TYPE ST_CoordinateGantryAxisEnable :
STRUCT
    {attribute 'pytmc' := '
        pv: bEnable
        io: i
        field: DESC Set false to prevent this function block from allowing the motors to enable.
    '}
    bEnable: BOOL; // Set false to prevent this function block from allowing the motors to enable.
    {attribute 'pytmc' := '
        pv: bLeaderDriveReady
        io: i
        field: DESC Intended to be linked to the leader drive ready status.
    '}
    bLeaderDriveReady AT %I*: BOOL; // Intended to be linked to the leader drive ready status.
    {attribute 'pytmc' := '
        pv: bFollowDriveReady
        io: i
        field: DESC Intended to be linked to the follow drive ready status.
    '}
    bFollowDriveReady AT %I*: BOOL; // Intended to be linked to the follow drive ready status.
    tTimeout: TIME := T#5s; // Timeout before giving up on a state.
    {attribute 'pytmc' := '
        pv: eState
        io: i
        field: DESC Present enable sequence state.
    '}
    eState: E_GantryEnableState; // Present enable sequence state.
END_STRUCT
END_TYPE

// ---- DUTs/ST_GarageSlot.TcDUT

TYPE ST_GarageSlot EXTENDS ST_SampleSlot :
(*
    Represents a slot in the SDS garage.
*)
STRUCT
    {attribute 'pytmc' := '
        pv: fYPos
        io: io
        field: DESC The y-position of the garage, in units of mm, which corresponds to the slot being approximately level with the transfer arm.
    '}
    fYPos: REAL;
    {attribute 'pytmc' := '
        pv: fDeg
        io: io
        field: DESC The angular position of the slot in the garage in units of degrees.
    '}
    fDeg: REAL;
END_STRUCT
END_TYPE

// ---- DUTs/ST_BoundedValue.TcDUT

TYPE ST_BoundedValue :
STRUCT
    {attribute 'pytmc' := '
        pv: fIn
        io: io
        field: DESC The input value before bounds are applied.
    '}
    fIn    : LREAL; // The input value before bounds are applied.
    {attribute 'pytmc' := '
        pv: fMax
        io: io
        field: DESC The maximum bound for the output value.
    '}
    fMax   : LREAL; // The maximum bound for the output value.
    {attribute 'pytmc' := '
        pv: fMin
        io: io
        field: DESC The minimum bound for the output value.
    '}
    fMin   : LREAL; // The minimum bound for the output value.
    {attribute 'pytmc' := '
        pv: fOut
        io: i
        field: DESC The output value after bounds are applied.
    '}
    fOut   : LREAL; // The output value after bounds are applied.
    {attribute 'pytmc' := '
        pv: bMaxLim
        io: i
        field: DESC TRUE if the output value has been limited by the upper bound.
    '}
    bMaxLim: BOOL; // TRUE if the output value has been limited by the upper bound.
    {attribute 'pytmc' := '
        pv: bMinLim
        io: i
        field: DESC TRUE if the output value has been limited by the lower bound.
    '}
    bMinLim: BOOL; // TRUE if the output value has been limited by the lower bound.
END_STRUCT
END_TYPE

// ---- DUTs/ST_DiffractometerSlot.TcDUT

TYPE ST_DiffractometerSlot EXTENDS ST_SampleSlot :
(*
    Represents a slot in the SDS garage.
*)
STRUCT
    {attribute 'pytmc' := '
        pv: fYPos
        io: io
        field: DESC The y-position of the garage, in units of mm, which corresponds to the slot being approximately level with the transfer arm.
    '}
    fYPos: REAL;
    {attribute 'pytmc' := '
        pv: fDeg
        io: io
        field: DESC The angular position of the slot in the garage in units of degrees.
    '}
    fDeg: REAL;
END_STRUCT
END_TYPE

// ---- DUTs/ST_MultiLeaderMotionCoupling.TcDUT

TYPE ST_MultiLeaderMotionCoupling :
STRUCT
    {attribute 'pytmc' := '
        pv: bEnable
        io: io
        field: DESC Set and hold TRUE to allow the axis to run in multi-leader mode.
    '}
    bEnable: BOOL;

    {attribute 'pytmc' := '
        pv: bReset
        io: io
        field: DESC Set and release TRUE to fully reset errors and state machine.
    '}
    bReset: BOOL;

    {attribute 'pytmc' := '
        pv: bBusy
        io: i
        field: DESC TRUE indicates state machine running and not in error state.
    '}
    bBusy: BOOL;

    {attribute 'pytmc' := '
        pv: sStatusMsg
        io: i
        field: DESC String used to give helpful messages.
    '}
    sStatusMsg: T_MaxString;

    // Ex: TIID^Device 2 (EtherCAT)^B950-233-WALL-S-R01-DRL-01^EL7047_02_11^STM Status^Status^Ready
    {attribute 'pytmc' := '
        pv: bFollowerDriveReady
        io: i
        field: DESC Linked to the ready status of the drive.
    '}
    bFollowerDriveReady AT %I*: BOOL; // Link to the ready status of the drive

    {attribute 'pytmc' := '
        pv: bUseDynamicLimits
        io: io
        field: DESC Set AND hold TRUE to enable dynamic limits to acc, vel, AND pos.
    '}
    bUseDynamicLimits: BOOL;

    {attribute 'pytmc' := '
        pv: fTargetAcc
        io: io
        field: DESC The target acceleration.
    '}
    fTargetAcc: LREAL; // Set in software to allow axis to target an acceleration based on multiple leaders.

    {attribute 'pytmc' := '
        pv: fTargetVel
        io: io
        field: DESC The target velocity.
    '}
    fTargetVel: LREAL; // Set in software to allow axis to target a velocity based on multiple leaders.

    {attribute 'pytmc' := '
        pv: fTargetPos
        io: io
        field: DESC The target position.
    '}
    fTargetPos: LREAL; // Set in software to allow axis to target a position based on multiple leaders.

    {attribute 'pytmc' := '
        pv: fPosDelta
        io: i
        field: DESC Target position minus position.
    '}
    fPosDelta : LREAL; // Difference between current position and target position.

    {attribute 'pytmc' := '
        pv: fTTGain
        io: io
        field: DESC Target tracking gain.
    '}
    fTargetTrackingGain: LREAL := 1; // Gain used to tune target tracking when within target position window.

    {attribute 'pytmc' := '
        pv: fHaltPos
        io: i
        field: DESC Position at which axis halted.
    '}
    fHaltPos: LREAL; // Position at which halt is called. Allows for centering deadband.

    {attribute 'pytmc' := 'pv: stAcc'}
    stAcc: ST_BoundedValue;

    {attribute 'pytmc' := 'pv: stVel'}
    stVel: ST_BoundedValue;

    {attribute 'pytmc' := 'pv: stPos'}
    stPos: ST_BoundedValue;

    {attribute 'pytmc' := '
        pv: nDir
        io: i
        field: DESC Internally calculated direction value for external setpoint generator.
    '}
    nDir: DINT;

    {attribute 'pytmc' := '
        pv: bError
        io: i
        field: DESC TRUE if an error is active.
    '}
    bError: BOOL;

    {attribute 'pytmc' := '
        pv: sErrorMsg
        io: i
        field: DESC Displays error message relevant to the active error. Empty otherwise.
    '}
    sErrorMsg: T_MaxString;

    {attribute 'pytmc' := '
        pv: sErrorHelp
        io: i
        field: DESC Displays additional help for the active rror. Empty otherwise.
    '}
    sErrorHelp: T_MaxString;

    {attribute 'pytmc' := '
        pv: eState
        io: i
        field: DESC Records the current state of the multi-leader function block.
    '}
    eState: E_MultiLeaderMotionCoupling;
END_STRUCT
END_TYPE

// ---- DUTs/ST_SampleSlot.TcDUT

TYPE ST_SampleSlot :
(*
    Represents a general slot for a sample puck.
*)
STRUCT
    {attribute 'pytmc' := '
        pv: eState
        io: io
        field: DESC Enumeration of possible states for a slot in the sample delivery system. (empty, full, or disabled)
    '}
    eState: E_SampleSlotStates;
    {attribute 'pytmc' := '
        pv: sTag
        io: i
        field: DESC A two character identifier for the slot. e.g., T1, B3, etc...
    '}
    sTag: STRING;
    {attribute 'pytmc' := '
        pv: sDesc
        io: io
        field: DESC If the slot is in the full state, this value is supposed to describe what is in the slot.
    '}
    sDesc: T_MaxString;
END_STRUCT
END_TYPE

// ---- DUTs/ST_SDS.TcDUT

TYPE ST_SDS :
(*
    Structure to represent the data used for the sample delivery system that is not
    needed to be persistent.
*)
STRUCT
    {attribute 'pytmc' := '
        pv: Initialized
        io: i
        field: DESC TRUE if the non-persistent data has been initialized. FALSE if it has not.
    '}
    bInitialized: BOOL;

    {attribute 'pytmc' := '
        pv: Enable
        io: io
        field: DESC TRUE to enable SDS system. FALSE to disable.
    '}
    bEnable : BOOL := TRUE;

    {attribute 'pytmc' := '
        pv: Maint
        io: io
        field: DESC TRUE if in maintenance mode. FALSE if NOT.
    '}
    bMaint: BOOL;

    {attribute 'pytmc' := '
        pv: Error
        io: i
        field: DESC TRUE if an error is active. FALSE if not.
    '}
    bError : BOOL;

    {attribute 'pytmc' := '
        pv: ErrorMsg
        io: i
        field: DESC Error message to help describe the active error.
    '}
    sErrorMsg : T_MaxString;

    {attribute 'pytmc' := '
        pv: Success
        io: i
        field: DESC TRUE if successfully completed state machine step.
    '}
    bSuccess : BOOL;

    // Variables used for homing
    {attribute 'pytmc' := '
        pv: HomeReq
        io: i
        field: DESC TRUE if homing is required for the sample transfer arm.
    '}
    bHomingRequired : BOOL := TRUE;
    tHomingRequiredTimeoutTime : TIME := T#1h;
    tonHomingRequiredTimeout : TON;
    tonHomingStateTimeout : TON;
    nHomingState : INT := 0;
    {attribute 'pytmc' := '
        pv: MinHomeReq
        io: i
        field: DESC Minutes until homing is required again for the sample transfer arm.
    '}
    fMinUntilHomingRequired: REAL;

    {attribute 'pytmc' := '
        pv: FaceState
        io: i
        field: DESC Enum to describe which way the sample garage should face.
    '}
    eFaceState: E_SDSFaceState;

    {attribute 'pytmc' := '
        pv: FacePortOffset
        io: io
        field: DESC Degree offset when trying to face the side port.
    '}
    fFacePortOffset: REAL := 90; // degree offset when trying to face the side port.

    // Transfer Arm State Positioner
    stTransferArmHEpicsToPlc: ST_StateEpicsToPlc;
    stTransferArmHPlcToEpics: ST_StatePlcToEpics;

    {attribute 'pytmc' := '
      pv: ArmHStateGet
      io: i
    '}
    eTransferArmHStateGet: E_SDSTransferArmHStates; // get state enum for transfer arm horizontal position states.

    {attribute 'pytmc' := '
      pv: ArmHStateSet
      io: io
    '}
    eTransferArmHStateSet: E_SDSTransferArmHStates; // set state enum for transfer arm horizontal position states.

    astTransferArmHPosState: ARRAY[1..GeneralConstants.MAX_STATES] OF ST_PositionState;
    {attribute 'pytmc' := '
        pv: ARMH:PS1D
        field: DESC Position State 1D used for transfer arm horizontal position states.
    '}
    fbTransferArmHPos1D: FB_PositionState1D; // Position State 1D used for transfer arm horizontal position states.

    // Transfer Arm State Positioner
    stTransferArmREpicsToPlc: ST_StateEpicsToPlc;
    stTransferArmRPlcToEpics: ST_StatePlcToEpics;

    {attribute 'pytmc' := '
      pv: ArmRStateGet
      io: i
    '}
    eTransferArmRStateGet: E_SDSTransferArmRStates; // get state enum for transfer arm rotational position states.

    {attribute 'pytmc' := '
      pv: ArmRStateSet
      io: io
    '}
    eTransferArmRStateSet: E_SDSTransferArmRStates; // set state enum for transfer arm rotational position states.

    astTransferArmRPosState: ARRAY[1..GeneralConstants.MAX_STATES] OF ST_PositionState;
    {attribute 'pytmc' := '
        pv: ARMR:PS1D
        field: DESC Position State 1D used for transfer arm rotational position states.
    '}
    fbTransferArmRPos1D: FB_PositionState1D; // Position State 1D used for transfer arm rotational position states.

    // Garage Y State Positioner
    stGarageYEpicsToPlc: ST_StateEpicsToPlc;
    stGarageYPlcToEpics: ST_StatePlcToEpics;

    {attribute 'pytmc' := '
      pv: GarYStateGet
      io: i
    '}
    eGarageYStateGet: E_SDSGarageYStates; // get state enum for garage y and rotational position states.

    {attribute 'pytmc' := '
      pv: GarYStateSet
      io: io
    '}
    eGarageYStateSet: E_SDSGarageYStates; // set state enum for garage y and rotational position states.

    astGarageYPosState: ARRAY[1..GeneralConstants.MAX_STATES] OF ST_PositionState;

    {attribute 'pytmc' := '
        pv: GARY:PS1D
        field: DESC Position State 1D used for garage y-position.
    '}
    fbGarageYPos1D: FB_PositionState1D; // Position State 1D used for garage y-position.

    // Garage R State Positioner
    stGarageREpicsToPlc: ST_StateEpicsToPlc;
    stGarageRPlcToEpics: ST_StatePlcToEpics;

    {attribute 'pytmc' := '
      pv: GarRStateGet
      io: i
    '}
    eGarageRStateGet: E_SDSGarageRStates; // get state enum for garage y and rotational position states.

    {attribute 'pytmc' := '
      pv: GarRStateSet
      io: io
    '}
    eGarageRStateSet: E_SDSGarageRStates; // set state enum for garage y and rotational position states.

    astGarageRPosState: ARRAY[1..GeneralConstants.MAX_STATES] OF ST_PositionState;

    {attribute 'pytmc' := '
        pv: GARR:PS1D
        field: DESC Position State 1D used for garage rotation..
    '}
    fbGarageRPos1D: FB_PositionState1D; // Position State 1D used for garage rotation.

    {attribute 'pytmc' := '
        pv: State
        field: DESC Present state for sample delivery system.
    '}
    eState : E_SDSState;

    {attribute 'pytmc' := '
        pv: SubState
        field: DESC Present sub-state for sample delivery system.
    '}
    eSubState : E_SDSSubState;

    {attribute 'pytmc' := '
        pv: SeqState
        field: DESC Present sequence state for sample delivery system.
    '}
    eSeqState: E_SDSSeqState;

    {attribute 'pytmc' := '
        pv: SecRemaining
        field: DESC Seconds remaining before current sequence step times out.
    '}
    fSecRemaining: REAL;

    {attribute 'pytmc' := '
        pv: StatusMsg
        field: DESC Status message.
    '}
    sStatusMsg: T_MaxString;

    // Booleans to track what is currently possible to do.

    {attribute 'pytmc' := '
        pv: GarLoadable
        io: i
        field: DESC True if it is currently possible to load a garage slot. False if all garage slots are full or disabled.
    '}
    bGarageLoadable : BOOL;

    {attribute 'pytmc' := '
        pv: GarUnloadable
        io: i
        field: DESC True if it is currently possible to unload a garage slot. False if all garage slots are empty or disabled.
    '}
    bGarageUnloadable : BOOL;

    {attribute 'pytmc' := '
        pv: ArmLoadable
        io: i
        field: DESC True if it is currently possible to load the transfer arm slot. False if the transfer arm slot is full or disabled.
    '}
    bTransferArmLoadable : BOOL;

    {attribute 'pytmc' := '
        pv: ArmUnloadable
        io: i
        field: DESC True if it is currently possible to unload the transfer arm slot. False if the transfer arm slot is empty or disabled.
    '}
    bTransferArmUnloadable : BOOL;

    {attribute 'pytmc' := '
        pv: DiffLoadable
        io: i
        field: DESC True if it is currently possible to load the diffractometer slot. False if the diffractometer slot is full or disabled.
    '}
    bDiffractometerLoadable : BOOL;

    {attribute 'pytmc' := '
        pv: DiffUnloadable
        io: i
        field: DESC True if it is currently possible to unload the diffractometer slot. False if the diffractoemter slot is empty or disabled.
    '}
    bDiffractometerUnloadable : BOOL;

    {attribute 'pytmc' := 'pv: Sel'}
    stUISelect : ST_UISelect;

    tonForwardHomingLimit: TON;

    stGarageYStage : REFERENCE TO ST_MotionStage;
    stGarageRStage : REFERENCE TO ST_MotionStage;
    stTransferArmHStage : REFERENCE TO ST_MotionStage;
    stTransferArmRStage : REFERENCE TO ST_MotionStage;

    eDiffXStateGet : REFERENCE TO E_DiffState;
    eDiffXStateSet : REFERENCE TO E_DiffState;
    stDiffXStage : REFERENCE TO ST_MotionStage;

    eDiffYStateGet : REFERENCE TO E_DiffState;
    eDiffYStateSet : REFERENCE TO E_DiffState;
    stDiffYStage : REFERENCE TO ST_MotionStage;

    eDiffZStateGet : REFERENCE TO E_DiffState;
    eDiffZStateSet : REFERENCE TO E_DiffState;
    stDiffZStage : REFERENCE TO ST_MotionStage;

    eDiff2ThetaYStateGet : REFERENCE TO E_DiffState;
    eDiff2ThetaYStateSet : REFERENCE TO E_DiffState;
    stDiff2ThetaYStage : REFERENCE TO ST_MotionStage;

    eDiffPhiStateGet : REFERENCE TO E_DiffState;
    eDiffPhiStateSet : REFERENCE TO E_DiffState;
    stDiffPhiStage : REFERENCE TO ST_MotionStage;

    eDiffChiStateGet : REFERENCE TO E_DiffState;
    eDiffChiStateSet : REFERENCE TO E_DiffState;
    stDiffChiStage : REFERENCE TO ST_MotionStage;

    eDiff2ThetaStateGet : REFERENCE TO E_DiffState;
    eDiff2ThetaStateSet : REFERENCE TO E_DiffState;
    stDiff2ThetaStage : REFERENCE TO ST_MotionStage;

    eDiffThetaStateGet : REFERENCE TO E_DiffState;
    eDiffThetaStateSet : REFERENCE TO E_DiffState;
    stDiffThetaStage : REFERENCE TO ST_MotionStage;

    {attribute 'pytmc' := '
        pv: GarAboveColl
        io: i
        field: DESC True if garage above collision height.
    '}
    bGarageAboveCollisionHeight : BOOL;

    {attribute 'pytmc' := '
        pv: TAHHomeState
        io: i
        field: DESC Transfer arm horizontal homing state.
    '}
    eTransferArmHHomingState : E_SDSHomingState;

    {attribute 'pytmc' := '
        pv: TARHomeState
        io: i
        field: DESC Transfer arm rotational homing state.
    '}
    eTransferArmRHomingState : E_SDSHomingState;

    {attribute 'pytmc' := '
        pv: GarRHomeState
        io: i
        field: DESC Garage rotational homing state.
    '}
    eGarageRHomingState : E_SDSHomingState;

    {attribute 'pytmc' := '
        pv: GarRotSpeed
        io: i
        field: DESC Garage rotational speed.
    '}
    fGarageRotationSpeed : LREAL := 10.0;

    {attribute 'pytmc' := '
        pv: TARotSpeed
        io: i
        field: DESC Garage rotational speed.
    '}
    fTransferArmRotationSpeed : LREAL := 10.0;

    {attribute 'pytmc' := '
        pv: GarRotClearancePos
        io: i
        field: DESC Garage rotational position to avoid collision with loaded transfer arm when moving up and down.
    '}
    fGarageRotationClearancePos : LREAL;

    {attribute 'pytmc' := '
        pv: LoadingSel
        io: i
        field: DESC True if loading from port.
    '}
    bLoadingSelected : BOOL;

    {attribute 'pytmc' := '
        pv: UnloadingSel
        io: i
        field: DESC True if unloading from port.
    '}
    bUnloadingSelected : BOOL;

    {attribute 'pytmc' := '
        pv: NumGarSlots
        io: i
        field: DESC Number of garage sample slots.
    '}
    nGarageSlots : UINT := 12;

    {attribute 'pytmc' := '
        pv: SelGarSlot
        io: i
        field: DESC Selected garage slot for loading/unloading.
    '}
    eSelectedGarageSlot : E_SDSGarageYStates;
END_STRUCT
END_TYPE

// ---- DUTs/ST_SDSPersistent.TcDUT

TYPE ST_SDSPersistent :
(*
    Structure to represent the data used for the sample delivery system that is
    needed to be persistent.
*)
STRUCT
    {attribute 'pytmc' := '
        pv: bInitialized
        io: i
        field: DESC TRUE if the persistent data has been initialized. FALSE if it has not.
    '}
    bInitialized: BOOL;

    {attribute 'pytmc' := 'pv: Garage:Slot'}
    astGarageSlot: ARRAY[E_SDSGarageYStates.T1..E_SDSGarageYStates.B4] OF ST_GarageSlot;

    {attribute 'pytmc' := 'pv: Transfer:Slot'}
    stTransferArmSlot: ST_TransferSlot;

    {attribute 'pytmc' := 'pv: Diff:Slot'}
    stDiffractometerSlot: ST_DiffractometerSlot;

    {attribute 'pytmc' := '
        pv: GarHSafeFromCol
        io: i
        field: DESC Height at which garage consider safe from collisions.
    '}
    fGarageHeightSafeFromCollision : LREAL := -10;

    {attribute 'pytmc' := '
        pv: GarRClearOff
        io: i
        field: DESC Garage rotational offset for clearance when moving up and down with loading transfer arm.
    '}
    fGarageRotationClearanceOffset : LREAL := 45;
END_STRUCT
END_TYPE

// ---- DUTs/ST_TransferSlot.TcDUT

TYPE ST_TransferSlot EXTENDS ST_SampleSlot :
(*
    Represents a slot in the SDS transfer arm.
*)
STRUCT
END_STRUCT
END_TYPE

// ---- DUTs/ST_UISelect.TcDUT

TYPE ST_UISelect :
STRUCT
    // Booleans to allow operator to choose what they want to do.
    {attribute 'pytmc' := '
        pv: Load
        io: io
        field: DESC Write True to command a loading sequence.
    '}
    bLoad: BOOL;

    {attribute 'pytmc' := '
        pv: Unload
        io: io
        field: DESC Write True to command a unloading sequence.
    '}
    bUnload: BOOL;

    {attribute 'pytmc' := '
        pv: ManualControl
        io: io
        field: DESC Write True to command manual control.
    '}
    bManualControl : BOOL;

    {attribute 'pytmc' := '
        pv: ExitManualControl
        io: io
        field: DESC Write True to command exit manual control.
    '}
    bExitManualControl : BOOL;

    {attribute 'pytmc' := '
        pv: LoadArmFromGar
        io: io
        field: DESC Write True to command load arm from garage.
    '}
    bLoadArmFromGarage : BOOL;

    {attribute 'pytmc' := '
        pv: UnloadArmToGar
        io: io
        field: DESC Write True to command unload arm from garage.
    '}
    bUnloadArmToGarage : BOOL;

    {attribute 'pytmc' := '
        pv: LoadGarFromPort
        io: io
        field: DESC Write True to command load garage from port.
    '}
    bLoadGarageFromPort : BOOL;

    {attribute 'pytmc' := '
        pv: UnloadGarFromPort
        io: io
        field: DESC Write True to command load garage from port.
    '}
    bLoadUnloadGarageFromPort : BOOL;

    {attribute 'pytmc' := '
        pv: LoadDiffFromArm
        io: io
        field: DESC Write True to command load diffractometer from arm.
    '}
    bLoadDiffractometerFromArm : BOOL;

    {attribute 'pytmc' := '
        pv: UnloadDiffToArm
        io: io
        field: DESC Write True to command unload diffractometer to arm.
    '}
    bUnloadDiffractometerToArm : BOOL;

    {attribute 'pytmc' := '
        pv: HomeArm
        io: io
        field: DESC Write True to command home transfer arm.
    '}
    bHomeTransferArm : BOOL;

    {attribute 'pytmc' := '
        pv: HomeGar
        io: io
        field: DESC Write True to command home garage.
    '}
    bHomeGarage : BOOL;

    {attribute 'pytmc' := '
        pv: GarSlot
        io: io
        field: DESC Select garage slot to unload or load.
    '}
    eGarageSlot : E_SDSGarageYStates;

    {attribute 'pytmc' := '
        pv: Proceed
        io: io
        field: DESC Write True to proceed to next sequence step, if applicable.
    '}
    bProceed: BOOL;

    {attribute 'pytmc' := '
        pv: Retry
        io: io
        field: DESC Write True when prompted to retry a defined previous step, if applicable.
    '}
    bRetry: BOOL;

    {attribute 'pytmc' := '
        pv: Cancel
        io: io
        field: DESC TRUE to cancel next sequence step.
    '}
    bCancel: BOOL;

    {attribute 'pytmc' := '
        pv: TextInput
        io: io
        field: DESC General purpose text input field.
    '}
    sTextInput: T_MaxString;
END_STRUCT
END_TYPE

// ---- Version/Global_Version.TcGVL
{attribute 'TcGenerated'}
{attribute 'no-analysis'}
{attribute 'linkalways'}
// This function has been automatically generated from the project information.
VAR_GLOBAL CONSTANT
    {attribute 'const_non_replaced'}
    stLibVersion_qrix_motion : ST_LibVersion := (iMajor := 0, iMinor := 4, iBuild := 0, iRevision := 0, nFlags := 1, sVersion := '0.4.0');
END_VAR

// ---- GVLs/GVL_EPS.TcGVL

VAR_GLOBAL
    {attribute 'pytmc' := 'pv: QRIX:SA:ESTOP_RST'}
    bResetIClk: BOOL;
    {attribute 'pytmc' := 'pv: QRIX:SA:ESTOP'}
    {attribute 'TcLinkTo' := 'TIIB[Rack#1A-02 SFIN (EL1918)]^StandardInputs^Standard Out Var 18'}
    bESTOP AT %I*: BOOL;

    {attribute 'TcLinkTo' := 'TIIB[Rack#2B-05 SV_AIR (EL2004)]^Channel 1^Output'}
    {attribute 'pytmc' := 'pv: QRIX:SA:SV1'}
    bOpenSV1 AT %Q*: BOOL;
    {attribute 'TcLinkTo' := 'TIIB[Rack#2B-05 SV_AIR (EL2004)]^Channel 2^Output'}
    {attribute 'pytmc' := 'pv: QRIX:SA:SV2'}
    bOpenSV2 AT %Q*: BOOL;

    {attribute 'TcLinkTo' := 'TIIB[Rack#1C_ServoDR (NCR-HD Series)]^260th receive PDO Mapping^Positive torque limit value'}
    iServoTorqueLimitPositive AT %Q*: UINT;

    {attribute 'TcLinkTo' := 'TIIB[Rack#1C_ServoDR (NCR-HD Series)]^260th receive PDO Mapping^Negative torque limit value'}
    iServoTorqueLimitNegative AT %Q*: UINT;

END_VAR

// ---- GVLs/GVL_Interface.TcGVL

{attribute 'qualified_only'}
VAR_GLOBAL

    (*I/O Outputs to QRIX Vacuum PLC*)

    {attribute 'TcLinkTo' :=  'TIID^Device 2 (EtherCAT)^B950-233-R03-DRL-01 (EK1200)^Term 141 (EL6692)^IO Outputs^QRIX_MOT_SDS_MMS_H_RAW_ENC_CNTS
    '}
    QRIX_MOT_SDS_MMS_H_RAW_ENC_CNTS AT %Q* : UINT;

    {attribute 'TcLinkTo' :=  'TIID^Device 2 (EtherCAT)^B950-233-R03-DRL-01 (EK1200)^Term 141 (EL6692)^IO Outputs^QRIX_MOT_SDS_MMS_H_FORWARD_EN
    '}
    QRIX_MOT_SDS_MMS_H_FORWARD_EN AT %Q* : BOOL;

    {attribute 'TcLinkTo' :=  'TIID^Device 2 (EtherCAT)^B950-233-R03-DRL-01 (EK1200)^Term 141 (EL6692)^IO Outputs^QRIX_MOT_SDS_MMS_H_BACKWARD_EN
    '}
    QRIX_MOT_SDS_MMS_H_BACKWARD_EN AT %Q* : BOOL;

    (*I/O Inputs from QRIX Vacuum PLC*)

    {attribute 'TcLinkTo' :=  'TIID^Device 2 (EtherCAT)^B950-233-R03-DRL-01 (EK1200)^Term 141 (EL6692)^IO Inputs^QRIX_VAC_VGC_03_OPEN_LIMIT_SWITCH
    '}
    QRIX_VAC_VGC_03_OPEN_LIMIT_SWITCH AT %I* : BOOL;

    {attribute 'TcLinkTo' :=  'TIID^Device 2 (EtherCAT)^B950-233-R03-DRL-01 (EK1200)^Term 141 (EL6692)^IO Inputs^QRIX_VAC_VGC_03_CLOSED_LIMIT_SWITCH
    '}
    QRIX_VAC_VGC_03_CLOSED_LIMIT_SWITCH AT %I* : BOOL;
    {attribute 'TcLinkTo' :=  'TIID^Device 2 (EtherCAT)^B950-233-R03-DRL-01 (EK1200)^Term 141 (EL6692)^IO Inputs^QRIX_VAC_VGC_03_OP_CMD
    '}
    QRIX_VAC_VGC_03_OP_CMD AT %I* : BOOL;

    {attribute 'TcLinkTo' :=  'TIID^Device 2 (EtherCAT)^B950-233-R03-DRL-01 (EK1200)^Term 141 (EL6692)^IO Inputs^QRIX_VAC_VGC_03_CL_CMD
    '}
    QRIX_VAC_VGC_03_CL_CMD AT %I* : BOOL;
END_VAR

// ---- GVLs/GVL_PMPS.TcGVL

{attribute 'qualified_only'}
VAR_GLOBAL
    {attribute 'pytmc' := 'pv: PLC:QRIX:MOTION:ARB'}
    fbArbiter: FB_Arbiter(1);
    {attribute 'pytmc' := 'pv: PLC:QRIX:MOTION:FFO:01'}
    {attribute 'TcLinkTo' := '.q_xFastFaultOut:=TIIB[PMPS_FFO]^Channel 1^Output'}
    fbFastFaultOutput1: FB_HardwareFFOutput := (bAutoReset := TRUE, i_sNetID:='172.21.92.73.1.1');
    {attribute 'pytmc' := 'pv: PLC:QRIX:MOTION:FFO:02'}
    {attribute 'TcLinkTo' := '.q_xFastFaultOut:=TIIB[PMPS_FFO]^Channel 2^Output'}
    fbFastFaultOutput2: FB_HardwareFFOutput := (bAutoReset := TRUE, i_sNetID:='172.21.92.73.1.1');
END_VAR

// ---- GVLs/GVL_Sensor.TcGVL

{attribute 'qualified_only'}
VAR_GLOBAL
    {attribute 'pytmc' := '
        pv: QRIX:SA:FLOATING
        io: i
    '}
    bFloating: BOOL;

    // YDF1
    {attribute 'pytmc' := '
        pv: QRIX:SA:DDS:YDF1
        io: i
    '}
    {attribute 'TcLinkTo' := '	.iRawCnts	:= TIIB[Rack#2D LinearGaugeAmp (SC-HG1-ETC)]^Process Data(In)  TxPDO-Map^Response Data Unit1'}
    stYDF1: DUT_SensorHGS;
    nYDF1 AT %Q*: UDINT;

    // YDF2
    {attribute 'pytmc' := '
        pv: QRIX:SA:DDS:YDF2
        io: i
    '}
    {attribute 'TcLinkTo' := '	.iRawCnts	:= TIIB[Rack#2D LinearGaugeAmp (SC-HG1-ETC)]^Process Data(In)  TxPDO-Map^Response Data Unit2'}
    stYDF2: DUT_SensorHGS;
    nYDF2 AT %Q*: UDINT;

    // YDF3
    {attribute 'pytmc' := '
        pv: QRIX:SA:DDS:YDF3
        io: i
    '}
    {attribute 'TcLinkTo' := '	.iRawCnts	:= TIIB[Rack#2D LinearGaugeAmp (SC-HG1-ETC)]^Process Data(In)  TxPDO-Map^Response Data Unit3'}
    stYDF3: DUT_SensorHGS;
    nYDF3 AT %Q*: UDINT;

    // Height difference btw granite shelf and detector frame.
    {attribute 'pytmc' := '
        pv: QRIX:SA:DDS:HDF
        io: i
    '}
    {attribute 'TcLinkTo' := '	.iRawCnts	:= TIIB[Rack#2D LinearGaugeAmp (SC-HG1-ETC)]^Process Data(In)  TxPDO-Map^Response Data Unit4'}
    stHDF: DUT_SensorHGS;

    // Granite TiltZ : Pitch
    {attribute 'pytmc' := '
        pv: QRIX:GS:INM:Z
        io: i
    '}
    {attribute 'TcLinkTo' := '	.iRawCnts	:= TIIB[Rack#2B-03 AI_TiltSensor (EL3174-0002)]^AI Standard Channel 2^Value'}
    stGraniteP: DUT_Sensor;
    // Granite TiltX : Roll
    {attribute 'pytmc' := '
        pv: QRIX:GS:INM:X
        io: i
    '}
    {attribute 'TcLinkTo' := '	.iRawCnts	:= TIIB[Rack#2B-03 AI_TiltSensor (EL3174-0002)]^AI Standard Channel 1^Value'}
    stGraniteR: DUT_Sensor;
    // Frame TiltZ : Pitch
    {attribute 'pytmc' := '
        pv: QRIX:DF:INM:Z
        io: i
    '}
    {attribute 'TcLinkTo' := '	.iRawCnts	:= TIIB[Rack#2B-03 AI_TiltSensor (EL3174-0002)]^AI Standard Channel 4^Value'}
    stFrameP: DUT_Sensor;
    // Frame TiltX : Roll
    {attribute 'pytmc' := '
        pv: QRIX:DF:INM:X
        io: i
    '}
    {attribute 'TcLinkTo' := '	.iRawCnts	:= TIIB[Rack#2B-03 AI_TiltSensor (EL3174-0002)]^AI Standard Channel 3^Value'}
    stFrameR: DUT_Sensor;

    {attribute 'pytmc' := '
        pv: QRIX:SA:GPT:PS1
        io: i
    '}
    {attribute 'TcLinkTo' := '	.iRawCnts	:= TIIB[Rack#2B-04 PS_P (EL3064)]^AI Standard Channel 1^Value'}
    stPS1: DUT_Sensor;
    {attribute 'pytmc' := '
        pv: QRIX:SA:GPT:PS2
        io: i
    '}
    {attribute 'TcLinkTo' := '	.iRawCnts	:= TIIB[Rack#2B-04 PS_P (EL3064)]^AI Standard Channel 2^Value'}
    stPS2: DUT_Sensor;
    {attribute 'pytmc' := '
        pv: QRIX:SA:GPT:PS3
        io: i
    '}
    {attribute 'TcLinkTo' := '	.iRawCnts	:= TIIB[Rack#2B-04 PS_P (EL3064)]^AI Standard Channel 3^Value'}
    stPS3: DUT_Sensor;
END_VAR

// ---- GVLs/GVL_VAR.TcGVL

VAR_GLOBAL

    {attribute 'pytmc' := '
        pv: QRIX:SA:bDoneJackOff
        io: i
    '}
    bDoneJackOff: BOOL;
    {attribute 'pytmc' := '
        pv: QRIX:SA:bDoneLevitation
        io: i
    '}
    bDoneLevitation: BOOL;
    {attribute 'pytmc' := '
        pv: QRIX:SA:bDoneLanding
        io: i
    '}
    bDoneLanding: BOOL;
    {attribute 'pytmc' := '
        pv: QRIX:SA:bDoneAdjustingRoll
        io: i
    '}
    bDoneAdjustingRoll: BOOL;
    {attribute 'pytmc' := '
        pv: QRIX:SA:bDoneAdjustingPitch
        io: i
    '}
    bDoneAdjustingPitch: BOOL;
    {attribute 'pytmc' := '
        pv: QRIX:SA:bDoneAdjustingHeight
        io: i
    '}
    bDoneAdjustingHeight: BOOL;

    // Reset and monitor circuit breakers on spectrometer arm
    // BOX0108 Circuit Breaker
    {attribute 'pytmc' := '
        pv: QRIX:SA:CB:B0108:Reset
        io: io
    '}
    {attribute 'TcLinkTo' := 'TIID^Device 2 (EtherCAT)^BOX-01 Coupler (EK1100)^BOX-08 CP_SDC (EL9221-5000)^OCP Outputs^Control^Reset'}
    bCircuitBreakerB0108Reset AT %Q*: BOOL;
    {attribute 'pytmc' := '
        pv: QRIX:SA:CB:B0108:Tripped
        io: i
    '}
    {attribute 'TcLinkTo' := 'TIID^Device 2 (EtherCAT)^BOX-01 Coupler (EK1100)^BOX-08 CP_SDC (EL9221-5000)^OCP Inputs^Status^Tripped'}
    bCircuitBreakerB0108Tripped AT %I*: BOOL;
    // BOX0113 Circuit Breaker
    {attribute 'pytmc' := '
        pv: QRIX:SA:CB:B0113:Reset
        io: io
    '}
    {attribute 'TcLinkTo' := 'TIID^Device 2 (EtherCAT)^BOX-01 Coupler (EK1100)^BOX-13 CP_DC (EL9221-5000)^OCP Outputs^Control^Reset'}
    bCircuitBreakerB0113Reset AT %Q*: BOOL;
    {attribute 'pytmc' := '
        pv: QRIX:SA:CB:B0113:Tripped
        io: i
    '}
    {attribute 'TcLinkTo' := 'TIID^Device 2 (EtherCAT)^BOX-01 Coupler (EK1100)^BOX-13 CP_DC (EL9221-5000)^OCP Inputs^Status^Tripped'}
    bCircuitBreakerB0113Tripped AT %I*: BOOL;
    // BOX0118 Circuit Breaker
    {attribute 'pytmc' := '
        pv: QRIX:SA:CB:B0118:Reset
        io: io
    '}
    {attribute 'TcLinkTo' := 'TIID^Device 2 (EtherCAT)^BOX-01 Coupler (EK1100)^BOX-18 CP_YF1_YF2 (EL9221-5000)^OCP Outputs^Control^Reset'}
    bCircuitBreakerB0118Reset AT %Q*: BOOL;
    {attribute 'pytmc' := '
        pv: QRIX:SA:CB:B0118:Tripped
        io: i
    '}
    {attribute 'TcLinkTo' := 'TIID^Device 2 (EtherCAT)^BOX-01 Coupler (EK1100)^BOX-18 CP_YF1_YF2 (EL9221-5000)^OCP Inputs^Status^Tripped'}
    bCircuitBreakerB0118Tripped AT %I*: BOOL;
    // Rack 2A02 Circuit Breaker
    {attribute 'pytmc' := '
        pv: QRIX:SA:CB:R2A02:Reset
        io: io
    '}
    {attribute 'TcLinkTo' := 'TIID^Device 2 (EtherCAT)^Rack#2A-01 Coupler (EK1100)^Rack#2A-02 CP_SLIT (EL9221-5000)^OCP Outputs^Control^Reset'}
    bCircuitBreakerR2A02Reset AT %Q*: BOOL;
    {attribute 'pytmc' := '
        pv: QRIX:SA:CB:R2A02:Tripped
        io: i
    '}
    {attribute 'TcLinkTo' := 'TIID^Device 2 (EtherCAT)^Rack#2A-01 Coupler (EK1100)^Rack#2A-02 CP_SLIT (EL9221-5000)^OCP Inputs^Status^Tripped'}
    bCircuitBreakerR2A02Tripped AT %I*: BOOL;
    // Rack 2A07 Circuit Breaker
    {attribute 'pytmc' := '
        pv: QRIX:SA:CB:R2A07:Reset
        io: io
    '}
    {attribute 'TcLinkTo' := 'TIID^Device 2 (EtherCAT)^Rack#2A-01 Coupler (EK1100)^Rack#2A-07 CP_G (EL9221-5000)^OCP Outputs^Control^Reset'}
    bCircuitBreakerR2A07Reset AT %Q*: BOOL;
    {attribute 'pytmc' := '
        pv: QRIX:SA:CB:R2A07:Tripped
        io: i
    '}
    {attribute 'TcLinkTo' := 'TIID^Device 2 (EtherCAT)^Rack#2A-01 Coupler (EK1100)^Rack#2A-07 CP_G (EL9221-5000)^OCP Inputs^Status^Tripped'}
    bCircuitBreakerR2A07Tripped AT %I*: BOOL;
    // Rack 2A13 Circuit Breaker
    {attribute 'pytmc' := '
        pv: QRIX:SA:CB:R2A13:Reset
        io: io
    '}
    {attribute 'TcLinkTo' := 'TIID^Device 2 (EtherCAT)^Rack#2A-01 Coupler (EK1100)^Rack#2A-13 CP_PM (EL9221-5000)^OCP Outputs^Control^Reset'}
    bCircuitBreakerR2A13Reset AT %Q*: BOOL;
    {attribute 'pytmc' := '
        pv: QRIX:SA:CB:R2A13:Tripped
        io: i
    '}
    {attribute 'TcLinkTo' := 'TIID^Device 2 (EtherCAT)^Rack#2A-01 Coupler (EK1100)^Rack#2A-13 CP_PM (EL9221-5000)^OCP Inputs^Status^Tripped'}
    bCircuitBreakerR2A13Tripped AT %I*: BOOL;
    // Rack 2B14 Circuit Breaker
    {attribute 'pytmc' := '
        pv: QRIX:SA:CB:R2B14:Reset
        io: io
    '}
    {attribute 'TcLinkTo' := 'TIID^Device 2 (EtherCAT)^Rack#2B-01 Coupler (EK1100)^Rack#2B-14 CP_YDF (EL9221-5000)^OCP Outputs^Control^Reset'}
    bCircuitBreakerR2B14Reset AT %Q*: BOOL;
    {attribute 'pytmc' := '
        pv: QRIX:SA:CB:R2B14:Tripped
        io: i
    '}
    {attribute 'TcLinkTo' := 'TIID^Device 2 (EtherCAT)^Rack#2B-01 Coupler (EK1100)^Rack#2B-14 CP_YDF (EL9221-5000)^OCP Inputs^Status^Tripped'}
    bCircuitBreakerR2B14Tripped AT %I*: BOOL;
    // Rack 2B17 Circuit Breaker
    {attribute 'pytmc' := '
        pv: QRIX:SA:CB:R2B17:Reset
        io: io
    '}
    {attribute 'TcLinkTo' := 'TIID^Device 2 (EtherCAT)^Rack#2B-01 Coupler (EK1100)^Rack#2B-17 CP_YDF_ZF (EL9221-5000)^OCP Outputs^Control^Reset'}
    bCircuitBreakerR2B17Reset AT %Q*: BOOL;
    {attribute 'pytmc' := '
        pv: QRIX:SA:CB:R2B17:Tripped
        io: i
    '}
    {attribute 'TcLinkTo' := 'TIID^Device 2 (EtherCAT)^Rack#2B-01 Coupler (EK1100)^Rack#2B-17 CP_YDF_ZF (EL9221-5000)^OCP Inputs^Status^Tripped'}
    bCircuitBreakerR2B17Tripped AT %I*: BOOL;

    fCryoZNeutralPositionAtDiffZ0 : LREAL;
    fCryoYNeutralPositionAtDiffY0 : LREAL;
    fBraidDiameter: LREAL := 70; // mm
END_VAR

// ---- GVLs/Main.TcGVL

{attribute 'qualified_only'}
VAR_GLOBAL

(*
    Only includes motor definitions for the IOC
    These are hard-coded to be Main.M#,
    but are very convenient to store in a GVL,
    hence the confusing namespace here
    This should be refactored once the IOC
    supports arbitrary ads paths for motors
*)
    // Sample Chamber Sliding Seal - 1 axis
    //connect EPS limits
    {attribute 'pytmc' := 'pv: QRIX:SC:SSL:MMS'}
    {attribute 'TcLinkTo' := '.bLimitForwardEnable  := TIIB[EL7047_02_01 - SSL]^STM Status^Status^Digital input 1;
                              .bLimitBackwardEnable := TIIB[EL7047_02_01 - SSL]^STM Status^Status^Digital input 2;
                              .nRawEncoderULINT     := TIIB[EL5042_02_02]^FB Inputs Channel 1^Position'}
    M1: ST_MotionStage := (sName := 'QRIX:SC:SSL:MMS');


    (* Start Adding Spectometer Arm Axes Here*)

    // 2Theta Stepper
    {attribute 'pytmc' := 'pv: QRIX:SA:MMS:2Theta'}
    {attribute 'TcLinkTo' := '	.bLimitForwardEnable  	:= TIIB[Rack#1A-04 DR_2Th (EL7047)]^STM Status^Status^Digital input 1;
                                .bLimitBackwardEnable 	:= TIIB[Rack#1A-04 DR_2Th (EL7047)]^STM Status^Status^Digital input 2;
                                .nRawEncoderULINT     	:= TIIB[Rack#1A-06 ENC_2Th (EL5042)]^FB Inputs Channel 1^Position;
                                .bBrakeRelease			:= TIIB[Rack#1A-05 MB_2Th (EL2602)]^Channel 1^Output
    '}
    M2: ST_MotionStage := (sName := 'QRIX:SA:MMS:2Theta');

    // XS1
    {attribute 'pytmc' := 'pv: QRIX:OPTSL:MMS:NORTH'}
    {attribute 'TcLinkTo' := '	.bLimitForwardEnable  	:= TIIB[Rack#2A-03 DR_XS1 (EL7041-0052)]^STM Status^Status^Digital input 1;
                                .bLimitBackwardEnable 	:= TIIB[Rack#2A-03 DR_XS1 (EL7041-0052)]^STM Status^Status^Digital input 2;
                                .nRawEncoderULINT     	:= TIIB[Rack#2B-07 ENC_X1_X2 (EL5042)]^FB Inputs Channel 1^Position
    '}
    M3: ST_MotionStage :=(sName := 'QRIX:OPTSL:MMS:NORTH');

    // XS2
    {attribute 'pytmc' := 'pv: QRIX:OPTSL:MMS:SOUTH'}
    {attribute 'TcLinkTo' := '	.bLimitForwardEnable  	:= TIIB[Rack#2A-04 DR_XS2 (EL7041-0052)]^STM Status^Status^Digital input 1;
                                .bLimitBackwardEnable 	:= TIIB[Rack#2A-04 DR_XS2 (EL7041-0052)]^STM Status^Status^Digital input 2;
                                .nRawEncoderULINT     	:= TIIB[Rack#2B-07 ENC_X1_X2 (EL5042)]^FB Inputs Channel 2^Position
    '}
    M4: ST_MotionStage:=(sName := 'QRIX:OPTSL:MMS:SOUTH');

    // YS1
    {attribute 'pytmc' := 'pv: QRIX:OPTSL:MMS:TOP'}
    {attribute 'TcLinkTo' := '	.bLimitForwardEnable  	:= TIIB[Rack#2A-05 DR_YS1 (EL7041-0052)]^STM Status^Status^Digital input 1;
                                .bLimitBackwardEnable 	:= TIIB[Rack#2A-05 DR_YS1 (EL7041-0052)]^STM Status^Status^Digital input 2;
                                .nRawEncoderULINT     	:= TIIB[Rack#2B-08 ENC_Y1_Y2 (EL5042)]^FB Inputs Channel 1^Position
    '}
    M5: ST_MotionStage:=(sName := 'QRIX:OPTSL:MMS:TOP');

    // YS2
    {attribute 'pytmc' := 'pv: QRIX:OPTSL:MMS:BOTTOM'}
    {attribute 'TcLinkTo' := '	.bLimitForwardEnable  	:= TIIB[Rack#2A-06 DR_YS2 (EL7041-0052)]^STM Status^Status^Digital input 1;
                                .bLimitBackwardEnable 	:= TIIB[Rack#2A-06 DR_YS2 (EL7041-0052)]^STM Status^Status^Digital input 2;
                                .nRawEncoderULINT     	:= TIIB[Rack#2B-08 ENC_Y1_Y2 (EL5042)]^FB Inputs Channel 1^Position
    '}
    M6: ST_MotionStage :=(sName := 'QRIX:OPTSL:MMS:BOTTOM');;

    // YG1
    {attribute 'pytmc' := 'pv: QRIX:OPT:MMS:Y1'}
    {attribute 'TcLinkTo' := '	.bLimitForwardEnable	:= TIIB[Rack#2A-10 DR_YG1 (EL7041-0052)]^STM Status^Status^Digital input 1;
                                .bLimitBackwardEnable	:= TIIB[Rack#2A-10 DR_YG1 (EL7041-0052)]^STM Status^Status^Digital input 2;
                                .nRawEncoderULINT		:= TIIB[Rack#2B-10 ENC_YG1_YG2 (EL5042)]^FB Inputs Channel 1^Position
    '}
    M7: ST_MotionStage:= (sName := 'QRIX:OPT:MMS:Y1');

    // YG2
    {attribute 'pytmc' := 'pv: QRIX:OPT:MMS:Y2'}
    {attribute 'TcLinkTo' := '	.bLimitForwardEnable	:= TIIB[Rack#2A-11 DR_YG2 (EL7041-0052)]^STM Status^Status^Digital input 1;
                                .bLimitBackwardEnable	:= TIIB[Rack#2A-11 DR_YG2 (EL7041-0052)]^STM Status^Status^Digital input 2;
                                .nRawEncoderULINT		:= TIIB[Rack#2B-10 ENC_YG1_YG2 (EL5042)]^FB Inputs Channel 2^Position
    '}
    M8: ST_MotionStage:= (sName := 'QRIX:OPT:MMS:Y2');

    // YG3
    {attribute 'pytmc' := 'pv: QRIX:OPT:MMS:Y3'}
    {attribute 'TcLinkTo' := '	.bLimitForwardEnable	:= TIIB[Rack#2A-12 DR_YG3 (EL7041-0052)]^STM Status^Status^Digital input 1;
                                .bLimitBackwardEnable	:= TIIB[Rack#2A-12 DR_YG3 (EL7041-0052)]^STM Status^Status^Digital input 2;
                                .nRawEncoderULINT		:= TIIB[Rack#2B-11 ENC_YG3_X1PM (EL5042)]^FB Inputs Channel 1^Position
    '}
    M9: ST_MotionStage:= (sName := 'QRIX:OPT:MMS:Y3');


    // RxG
    {attribute 'pytmc' := 'pv: QRIX:G:MMS:Rx'}
    {attribute 'TcLinkTo' := '	.bLimitForwardEnable	:= TIIB[Rack#2A-08 DR_RxG (EL7041-0052)]^STM Status^Status^Digital input 1;
                                .bLimitBackwardEnable	:= TIIB[Rack#2A-08 DR_RxG (EL7041-0052)]^STM Status^Status^Digital input 2;
                                .nRawEncoderULINT		:= TIIB[Rack#2B-09 ENC_RxG_XG (EL5042)]^FB Inputs Channel 1 compact^Position
    '}
    M10: ST_MotionStage:=(sName := 'QRIX:G:MMS:Rx');

    // XG
    {attribute 'pytmc' := 'pv: QRIX:G:MMS:X'}
    {attribute 'TcLinkTo' := '	.bLimitForwardEnable	:= TIIB[Rack#2A-09 DR_XG (EL7041-0052)]^STM Status^Status^Digital input 1;
                                .bLimitBackwardEnable	:= TIIB[Rack#2A-09 DR_XG (EL7041-0052)]^STM Status^Status^Digital input 2;
                                .nRawEncoderULINT		:= TIIB[Rack#2B-09 ENC_RxG_XG (EL5042)]^FB Inputs Channel 2^Position
    '}
    M11: ST_MotionStage:=(sName := 'QRIX:G:MMS:X');

    // XPM1
    {attribute 'pytmc' := 'pv: QRIX:PM:MMS:X1'}
    {attribute 'TcLinkTo' := '	.bLimitForwardEnable	:= TIIB[Rack#2A-14 DR_XPM1 (EL7041-0052)]^STM Status^Status^Digital input 1;
                                .bLimitBackwardEnable	:= TIIB[Rack#2A-14 DR_XPM1 (EL7041-0052)]^STM Status^Status^Digital input 2;
                                .nRawEncoderULINT		:= TIIB[Rack#2B-11 ENC_YG3_X1PM (EL5042)]^FB Inputs Channel 2^Position
    '}
    M12: ST_MotionStage :=(sName := 'QRIX:PM:MMS:X1');

    // XPM2
    {attribute 'pytmc' := 'pv: QRIX:PM:MMS:X2'}
    {attribute 'TcLinkTo' := '	.bLimitForwardEnable	:= TIIB[Rack#2A-15 DR_XPM2 (EL7041-0052)]^STM Status^Status^Digital input 1;
                                .bLimitBackwardEnable	:= TIIB[Rack#2A-15 DR_XPM2 (EL7041-0052)]^STM Status^Status^Digital input 2;
                                .nRawEncoderULINT		:= TIIB[Rack#2B-12 ENC_X2PM_RzPM (EL5042)]^FB Inputs Channel 1^Position
    '}
    M13: ST_MotionStage:=(sName := 'QRIX:PM:MMS:X2');

    // RzPM
    {attribute 'pytmc' := 'pv: QRIX:PM:MMS:Rz'}
    {attribute 'TcLinkTo' := '	.bLimitForwardEnable	:= TIIB[Rack#2A-16 DR_RzPM (EL7041-0052)]^STM Status^Status^Digital input 1;
                                .bLimitBackwardEnable	:= TIIB[Rack#2A-16 DR_RzPM (EL7041-0052)]^STM Status^Status^Digital input 2;
                                .nRawEncoderULINT		:= TIIB[Rack#2B-12 ENC_X2PM_RzPM (EL5042)]^FB Inputs Channel 2^Position
    '}
    M14: ST_MotionStage:=(sName := 'QRIX:PM:MMS:Rz');

    // YDF1
    {attribute 'pytmc' := 'pv: QRIX:DF:MMS:Y1'}
    {attribute 'TcLinkTo' := '	.bLimitForwardEnable  	:= TIIB[Rack#2B-15 DR_YDF1 (EL7041-0052)]^STM Status^Status^Digital input 1;
                                .bLimitBackwardEnable 	:= TIIB[Rack#2B-15 DR_YDF1 (EL7041-0052)]^STM Status^Status^Digital input 2;
                                .nRawEncoderULINT		:= TIID^Device 2 (EtherCAT)^Rack#2D LinearGaugeAmp (SC-HG1-ETC)^Process Data(In)  TxPDO-Map^Response Data Unit1
    '}
    M15: ST_MotionStage :=(sName := 'QRIX:DF:MMS:Y1');

    // YDF2
    {attribute 'pytmc' := 'pv: QRIX:DF:MMS:Y2'}
    {attribute 'TcLinkTo' := '	.bLimitForwardEnable  	:= TIIB[Rack#2B-16 DR_YDF2 (EL7041-0052)]^STM Status^Status^Digital input 1;
                                .bLimitBackwardEnable 	:= TIIB[Rack#2B-16 DR_YDF2 (EL7041-0052)]^STM Status^Status^Digital input 2;
                                .nRawEncoderULINT		:= TIID^Device 2 (EtherCAT)^Rack#2D LinearGaugeAmp (SC-HG1-ETC)^Process Data(In)  TxPDO-Map^Response Data Unit2
    '}
    M16: ST_MotionStage:=(sName := 'QRIX:DF:MMS:Y2');

    // YDF3
    {attribute 'pytmc' := 'pv: QRIX:DF:MMS:Y3'}
    {attribute 'TcLinkTo' := '	.bLimitForwardEnable  	:= TIIB[Rack#2B-19 DR_YDF3 (EL7041-0052)]^STM Status^Status^Digital input 1;
                                .bLimitBackwardEnable 	:= TIIB[Rack#2B-19 DR_YDF3 (EL7041-0052)]^STM Status^Status^Digital input 2;
                                .nRawEncoderULINT		:= TIID^Device 2 (EtherCAT)^Rack#2D LinearGaugeAmp (SC-HG1-ETC)^Process Data(In)  TxPDO-Map^Response Data Unit3
    '}
    M17: ST_MotionStage :=(sName := 'QRIX:DF:MMS:Y3');

    // XSDC1
    {attribute 'pytmc' := 'pv: QRIX:DETSL:MMS:NORTH'}
    {attribute 'TcLinkTo' := '	.bLimitForwardEnable  	:= TIIB[BOX-09 DR_XSDC1 (EL7041-0052)]^STM Status^Status^Digital input 1;
                                .bLimitBackwardEnable 	:= TIIB[BOX-09 DR_XSDC1 (EL7041-0052)]^STM Status^Status^Digital input 2;
                                .nRawEncoderULINT     	:= TIIB[BOX-03 ENC_X1_X2 (EL5042)]^FB Inputs Channel 1^Position
    '}
    M18: ST_MotionStage:=(sName := 'QRIX:DETSL:MMS:NORTH');

    // XSDC2
    {attribute 'pytmc' := 'pv: QRIX:DETSL:MMS:SOUTH'}
    {attribute 'TcLinkTo' := '	.bLimitForwardEnable	:= TIIB[BOX-10 DR_XSDC2 (EL7041-0052)]^STM Status^Status^Digital input 1;
                                .bLimitBackwardEnable 	:= TIIB[BOX-10 DR_XSDC2 (EL7041-0052)]^STM Status^Status^Digital input 2;
                                .nRawEncoderULINT     	:= TIIB[BOX-03 ENC_X1_X2 (EL5042)]^FB Inputs Channel 2^Position
    '}
    M19: ST_MotionStage :=(sName := 'QRIX:DETSL:MMS:SOUTH');

    // YSDC1
    {attribute 'pytmc' := 'pv: QRIX:DETSL:MMS:TOP'}
    {attribute 'TcLinkTo' := '	.bLimitForwardEnable	:= TIIB[BOX-11 DR_YSDC1 (EL7041-0052)]^STM Status^Status^Digital input 1;
                                .bLimitBackwardEnable 	:= TIIB[BOX-11 DR_YSDC1 (EL7041-0052)]^STM Status^Status^Digital input 2;
                                .nRawEncoderULINT     	:= TIIB[BOX-04 ENC_Y1_Y2 (EL5042)]^FB Inputs Channel 1^Position
    '}
    M20: ST_MotionStage :=(sName := 'QRIX:DETSL:MMS:TOP');

    // YSDC2
    {attribute 'pytmc' := 'pv: QRIX:DETSL:MMS:BOTTOM'}
    {attribute 'TcLinkTo' := '	.bLimitForwardEnable	:= TIIB[BOX-12 DR_YSDC2 (EL7041-0052)]^STM Status^Status^Digital input 1;
                                .bLimitBackwardEnable 	:= TIIB[BOX-12 DR_YSDC2 (EL7041-0052)]^STM Status^Status^Digital input 2;
                                .nRawEncoderULINT     	:= TIIB[BOX-04 ENC_Y1_Y2 (EL5042)]^FB Inputs Channel 1^Position
    '}
    M21: ST_MotionStage :=(sName := 'QRIX:DETSL:MMS:BOTTOM');

    // XDC
    {attribute 'pytmc' := 'pv: QRIX:DC:MMS:X'}
    {attribute 'TcLinkTo' := '	.bLimitForwardEnable  	:= TIIB[BOX-14 DR_XDC (EL7041-0052)]^STM Status^Status^Digital input 1;
                                .bLimitBackwardEnable 	:= TIIB[BOX-14 DR_XDC (EL7041-0052)]^STM Status^Status^Digital input 2;
                                .nRawEncoderULINT     	:= TIIB[BOX-05 ENC_XDC_RyDC (EL5042)]^FB Inputs Channel 1^Position
    '}
    M22: ST_MotionStage:=(sName := 'QRIX:DC:MMS:X');

    // RyDC
    {attribute 'pytmc' := 'pv: QRIX:DC:MMS:Ry'}
    {attribute 'TcLinkTo' := '	.bLimitForwardEnable	:= TIIB[BOX-15 DR_RyDC (EL7041-0052)]^STM Status^Status^Digital input 1;
                                .bLimitBackwardEnable	:= TIIB[BOX-15 DR_RyDC (EL7041-0052)]^STM Status^Status^Digital input 2;
                                .nRawEncoderULINT		:= TIIB[BOX-05 ENC_XDC_RyDC (EL5042)]^FB Inputs Channel 2^Position
    '}
    M23: ST_MotionStage :=(sName := 'QRIX:DC:MMS:Ry');

    // ZDC
    {attribute 'pytmc' := 'pv: QRIX:DC:MMS:Z'}
    {attribute 'TcLinkTo' := '	.bLimitForwardEnable	:= TIIB[BOX-16 DR_ZDC (EL7041-0052)]^STM Status^Status^Digital input 1;
                                .bLimitBackwardEnable	:= TIIB[BOX-16 DR_ZDC (EL7041-0052)]^STM Status^Status^Digital input 2;
                                .nRawEncoderULINT		:= TIIB[BOX-06 ENC_ZDC_YF1 (EL5042)]^FB Inputs Channel 1^Position
    '}
    M24: ST_MotionStage:=(sName := 'QRIX:DC:MMS:Z');

    // YF1
    {attribute 'pytmc' := 'pv: QRIX:DA:MMS:Y1'}
    {attribute 'TcLinkTo' := '	.bLimitForwardEnable	:= TIIB[Rack#1A-02 SFIN (EL1918)]^StandardInputs^Standard Out Var 10;
                                .bLimitBackwardEnable 	:= TIIB[Rack#1A-02 SFIN (EL1918)]^StandardInputs^Standard Out Var 11;
                                .nRawEncoderULINT     	:= TIIB[BOX-06 ENC_ZDC_YF1 (EL5042)]^FB Inputs Channel 2^Position;
                                .bBrakeRelease        	:= TIIB[BOX-19 MB_YF1_YF2 (EL2602)]^Channel 1^Output
    '}
    M25: ST_MotionStage:=(sName := 'QRIX:DA:MMS:Y1');

    // YF2
    {attribute 'pytmc' := 'pv: QRIX:DA:MMS:Y2'}
    {attribute 'TcLinkTo' := '	.bLimitForwardEnable	:= TIIB[Rack#1A-02 SFIN (EL1918)]^StandardInputs^Standard Out Var 12;
                                .bLimitBackwardEnable	:= TIIB[Rack#1A-02 SFIN (EL1918)]^StandardInputs^Standard Out Var 13;
                                .nRawEncoderULINT     	:= TIIB[BOX-07 ENC_YF2_ZF (EL5042)]^FB Inputs Channel 1^Position;
                                .bBrakeRelease			:= TIIB[BOX-19 MB_YF1_YF2 (EL2602)]^Channel 2^Output
    '}
    M26: ST_MotionStage:=(sName := 'QRIX:DA:MMS:Y2');

    // ZF
    {attribute 'pytmc' := 'pv: QRIX:DA:MMS:Z'}
    {attribute 'TcLinkTo' := '	.bLimitForwardEnable	:= TIIB[Rack#1A-02 SFIN (EL1918)]^StandardInputs^Standard Out Var 14;
                                .bLimitBackwardEnable	:= TIIB[Rack#1A-02 SFIN (EL1918)]^StandardInputs^Standard Out Var 15;
                                .nRawEncoderULINT		:= TIIB[BOX-07 ENC_YF2_ZF (EL5042)]^FB Inputs Channel 2^Position;
                                .bBrakeRelease			:= TIIB[Rack#2B-18 MB_ZF (EL2602)]^Channel 1^Output
    '}
    M27: ST_MotionStage:=(sName := 'QRIX:DA:MMS:Z');


    // Diffractometer -  8 axes START AT M28
    {attribute 'pytmc' := 'pv: QRIX:DIFF:MMS:X'}
    {attribute 'TcLinkTo' := '.bLimitForwardEnable  := TIIB[EL1088_03_04]^Channel 2^Input;
                              .bLimitBackwardEnable := TIIB[EL1088_03_04]^Channel 1^Input;
                              .bHome := TIIB[EL1088_03_10]^Channel 1^Input;
                              .nRawEncoderULINT     := TIIB[EL5042_03_02-Diff-X-Y]^FB Inputs Channel 1^Position'}
    M28: ST_MotionStage := (sName := 'QRIX:DIFF:MMS:X');

    {attribute 'pytmc' := 'pv: QRIX:DIFF:MMS:Y'}
    {attribute 'TcLinkTo' := '.bLimitForwardEnable  := TIIB[EL1088_03_04]^Channel 4^Input;
                              .bLimitBackwardEnable := TIIB[EL1088_03_04]^Channel 3^Input;
                              .bHome := TIIB[EL1088_03_10]^Channel 2^Input;
                              .nRawEncoderULINT     := TIIB[EL5042_03_02-Diff-X-Y]^FB Inputs Channel 2^Position'}
    M29: ST_MotionStage := (sName := 'QRIX:DIFF:MMS:Y');

    {attribute 'pytmc' := 'pv: QRIX:DIFF:MMS:Z'}
    {attribute 'TcLinkTo' := '.bLimitForwardEnable  := TIIB[EL1088_03_08]^Channel 2^Input;
                              .bLimitBackwardEnable := TIIB[EL1088_03_08]^Channel 1^Input;
                              .bHome := TIIB[EL1088_03_10]^Channel 3^Input;
                              .nRawEncoderULINT     := TIIB[EL5042_03_06-DIff-Z-2ThetaY]^FB Inputs Channel 1^Position'}
    M30: ST_MotionStage := (sName := 'QRIX:DIFF:MMS:Z');

    {attribute 'pytmc' := 'pv: QRIX:DIFF:MMS:DETY'}
    {attribute 'TcLinkTo' := '.bLimitForwardEnable  := TIIB[EL1088_03_08]^Channel 5^Input;
                              .bLimitBackwardEnable := TIIB[EL1088_03_08]^Channel 6^Input;
                              .bHome := TIIB[EL1088_03_10]^Channel 4^Input;
                              .nRawEncoderULINT     := TIIB[EL5042_03_06-DIff-Z-2ThetaY]^FB Inputs Channel 2^Position'}
    M31: ST_MotionStage := (sName := 'QRIX:DIFF:MMS:DETY');

    {attribute 'pytmc' := 'pv: QRIX:DIFF:MMS:PHI'}
    {attribute 'TcLinkTo' := '.bLimitForwardEnable  := TIIB[EL1088_03_08]^Channel 3^Input;
                              .bLimitBackwardEnable := TIIB[EL1088_03_08]^Channel 4^Input;
                              .bHome := TIIB[EL1088_03_10]^Channel 4^Input;
                              .nRawEncoderULINT     := TIIB[EL5042_03_13 - Diff - Phi - Chi]^FB Inputs Channel 1^Position'}
    M32: ST_MotionStage := (sName := 'QRIX:DIFF:MMS:PHI');

    {attribute 'pytmc' := 'pv: QRIX:DIFF:MMS:CHI'}
    {attribute 'TcLinkTo' := '.bLimitForwardEnable  := TIIB[EL1088_03_15]^Channel 2^Input;
                              .bLimitBackwardEnable := TIIB[EL1088_03_15]^Channel 1^Input;
                              .bHome := TIIB[EL1088_03_10]^Channel 6^Input;
                              .nRawEncoderULINT     := TIIB[EL5042_03_13 - Diff - Phi - Chi]^FB Inputs Channel 2^Position'}
    M33: ST_MotionStage := (sName := 'QRIX:DIFF:MMS:CHI');

    {attribute 'pytmc' := 'pv: QRIX:DIFF:MMS:THETA'}
    {attribute 'TcLinkTo' := '.bLimitForwardEnable  := TIIB[EL1088_03_15]^Channel 3^Input;
                              .bLimitBackwardEnable := TIIB[EL1088_03_15]^Channel 4^Input;
                              .bHome := TIIB[EL1088_03_10]^Channel 7^Input;
                              .nRawEncoderULINT     := TIIB[EL5042_03_17 - Diff - Theta - 2Theta]^FB Inputs Channel 1^Position'}
    M34: ST_MotionStage := (sName := 'QRIX:DIFF:MMS:THETA');

    {attribute 'pytmc' := 'pv: QRIX:DIFF:MMS:2THETA'}
    {attribute 'TcLinkTo' := '.bLimitForwardEnable  := TIIB[EL1088_03_15]^Channel 5^Input;
                              .bLimitBackwardEnable := TIIB[EL1088_03_15]^Channel 6^Input;
                              .bHome := TIIB[EL1088_03_10]^Channel 8^Input;
                              .nRawEncoderULINT     := TIIB[EL5042_03_17 - Diff - Theta - 2Theta]^FB Inputs Channel 2^Position'}
    M35: ST_MotionStage := (sName := 'QRIX:DIFF:MMS:2THETA');



    // Laser Table  -  3 axes
    {attribute 'pytmc' := 'pv: QRIX:LAS:MMS:VIS'}
    {attribute 'TcLinkTo' := '.bLimitForwardEnable  := TIIB[EL1088_02_06]^Channel 6^Input;
                              .bLimitBackwardEnable :=  TIIB[EL1088_02_06]^Channel 5^Input;
                              .nRawEncoderULINT     := TIIB[EL5042_02_05 - LAS_VIS]^FB Inputs Channel 1^Position'}
    M36: ST_MotionStage := (sName := 'QRIX:LAS:MMS:VIS');

    {attribute 'pytmc' := 'pv: QRIX:DIAG:MMS:H'}
    {attribute 'TcLinkTo' := '.bLimitForwardEnable  :=  TIIB[EL1088_02_06]^Channel 2^Input;
                              .bLimitBackwardEnable :=  TIIB[EL1088_02_06]^Channel 1^Input;
                              .nRawEncoderULINT     := TIIB[EL5042_02_08 - LAS_D_V-H]^FB Inputs Channel 2^Position'}
    M37: ST_MotionStage := (sName := 'QRIX:DIAG:MMS:H');

    {attribute 'pytmc' := 'pv: QRIX:DIAG:MMS:V'}
    {attribute 'TcLinkTo' := '.bLimitForwardEnable  := TIIB[EL1088_02_06]^Channel 4^Input;
                              .bLimitBackwardEnable := TIIB[EL1088_02_06]^Channel 3^Input;
                              .nRawEncoderULINT     := TIIB[EL5042_02_08 - LAS_D_V-H]^FB Inputs Channel 1^Position'}
    M38: ST_MotionStage := (sName := 'QRIX:DIAG:MMS:V');


    //Sample Delivery - 6 Axes


    {attribute 'pytmc' := 'pv: QRIX:SDS:MMS:X'}
    {attribute 'TcLinkTo' := '.bLimitForwardEnable  := TIIB[EL7047_04_01]^STM Status^Status^Digital input 1;
                              .bLimitBackwardEnable := TIIB[EL7047_04_01]^STM Status^Status^Digital input 2;
                              .nRawEncoderULINT     := TIIB[EL5042_04_02]^FB Inputs Channel 1^Position;
                              .bHome 				:= TIIB[EL1004_04_04]^Channel 1^Input'}
    M39: ST_MotionStage := (sName := 'QRIX:SDS:MMS:X');

    {attribute 'pytmc' := 'pv: QRIX:SDS:MMS:Y'}
    {attribute 'TcLinkTo' := '.bLimitForwardEnable  := TIIB[EL7047_04_03]^STM Status^Status^Digital input 2;
                              .bLimitBackwardEnable := TIIB[EL7047_04_03]^STM Status^Status^Digital input 1;
                              .nRawEncoderULINT     := TIIB[EL5042_04_02]^FB Inputs Channel 2^Position;
                              .bHome 				:= TIIB[EL1004_04_04]^Channel 2^Input'}
    M40: ST_MotionStage := (sName := 'QRIX:SDS:MMS:Y');

    {attribute 'pytmc' := 'pv: QRIX:SDS:MMS:Z'}
    {attribute 'TcLinkTo' := '.bLimitForwardEnable  := TIIB[EL7047_04_05]^STM Status^Status^Digital input 1;
                              .bLimitBackwardEnable := TIIB[EL7047_04_05]^STM Status^Status^Digital input 2;
                              .nRawEncoderULINT     := TIIB[EL5042_04_06]^FB Inputs Channel 1^Position;
                              .bHome 				:= TIIB[EL1004_04_04]^Channel 3^Input'}
    M41: ST_MotionStage := (sName := 'QRIX:SDS:MMS:Z');

     {attribute 'pytmc' := 'pv: QRIX:SDS:MMS:ROT_V'}
    {attribute 'TcLinkTo' := '.nRawEncoderUINT     := TIIB[EL5101_05_01]^ENC Status compact^Counter value;
                              .bHome 				:= TIIB[EL1004_04_04]^Channel 4^Input'}
    M42: ST_MotionStage := (sName := 'QRIX:SDS:MMS:ROT_V');

    {attribute 'pytmc' := 'pv: QRIX:SDS:MMS:ROT_H'}
    {attribute 'TcLinkTo' := '.bLimitForwardEnable  := TIIB[EL7047_04_10]^STM Status^Status^Digital input 2;
                              .bLimitBackwardEnable := TIIB[EL7047_04_10]^STM Status^Status^Digital input 1;
                              .nRawEncoderUINT     := TIIB[EL5101_05_02]^ENC Status compact^Counter value;
                              .bHome 				:= TIIB[EL1004_04_09]^Channel 1^Input'}
    M43: ST_MotionStage := (sName := 'QRIX:SDS:MMS:ROT_H');

    {attribute 'pytmc' := 'pv: QRIX:SDS:MMS:H'}
    {attribute 'TcLinkTo' := '.bLimitForwardEnable  := TIIB[EL7047_04_12]^STM Status^Status^Digital input 1;
                              .bLimitBackwardEnable := TIIB[EL7047_04_12]^STM Status^Status^Digital input 2;
                              .bHome 				:= TIIB[EL1004_04_09]^Channel 3^Input;
                              .nRawEncoderUINT     := TIIB[EL5101_05_03]^ENC Status compact^Counter value'}
    M44: ST_MotionStage := (sName := 'QRIX:SDS:MMS:H');

    //Detector Rotation
    {attribute 'pytmc' := 'pv: QRIX:DET:MMS:ROT'}
    {attribute 'TcLinkTo' := '.nRawEncoderULINT     := TIIB[BOX-22 DET_ROT (EL5042)]^FB Inputs Channel 1^Position'}
    M45: ST_MotionStage := (sName := 'QRIX:DET:MMS:ROT');

    // Cryo -  4 axes
    //Cryo -X
    {attribute 'pytmc' := 'pv: QRIX:CRYO:MMS:X'}
    {attribute 'TcLinkTo' := '.bLimitForwardEnable  := TIIB[EL7047_02_12]^STM Status^Status^Digital input 1;
                              .bLimitBackwardEnable := TIIB[EL7047_02_12]^STM Status^Status^Digital input 2;
                              .nRawEncoderULINT     := TIIB[EL5042_02_13]^FB Inputs Channel 1^Position'}
    M46: ST_MotionStage := (sName := 'QRIX:CRYO:MMS:X');
    //CRYO Y
    {attribute 'pytmc' := 'pv: QRIX:CRYO:MMS:Y'}
    {attribute 'TcLinkTo' := '.bLimitForwardEnable  := TIIB[EL7047_02_14]^STM Status^Status^Digital input 2;
                              .bLimitBackwardEnable := TIIB[EL7047_02_14]^STM Status^Status^Digital input 1;
                              .nRawEncoderULINT     := TIIB[EL5042_02_13]^FB Inputs Channel 2^Position'}
    M47: ST_MotionStage := (sName := 'QRIX:CRYO:MMS:Y');
    //CRYO Z
    {attribute 'pytmc' := 'pv: QRIX:CRYO:MMS:Z'}
    {attribute 'TcLinkTo' := '.bLimitForwardEnable  := TIIB[EL7047_02_15]^STM Status^Status^Digital input 1;
                              .bLimitBackwardEnable := TIIB[EL7047_02_15]^STM Status^Status^Digital input 2;
                              .nRawEncoderULINT     := TIIB[EL5042_02_16]^FB Inputs Channel 1^Position'}
    M48: ST_MotionStage := (sName := 'QRIX:CRYO:MMS:Z');
    // CRYO-ROT
    {attribute 'pytmc' := 'pv: QRIX:CRYO:MMS:ROT'}
    {attribute 'TcLinkTo' := '.nRawEncoderULINT     := TIIB[EL5042_02_16]^FB Inputs Channel 2^Position'}
    M49: ST_MotionStage := (sName := 'QRIX:CRYO:MMS:ROT');

(*
    // Questar -  2 axes
    {attribute 'pytmc' := 'pv: QRIX:QUESTAR:MMS:01'}
    {attribute 'TcLinkTo' := '.bLimitForwardEnable  := TIIB[SSL-EL7041]^STM Status^Status^Digital input 1;
                              .bLimitBackwardEnable := TIIB[SSL-EL7041]^STM Status^Status^Digital input 2;
                              .nRawEncoderULINT     := TIIB[IM1K3-EL5042]^FB Inputs Channel 1^Position'}
    M49: ST_MotionStage := (sName := 'QRIX:QUESTAR:MMS:01');

    {attribute 'pytmc' := 'pv: QRIX:QUESTAR:MMS:02'}
    {attribute 'TcLinkTo' := '.bLimitForwardEnable  := TIIB[SSL-EL7041]^STM Status^Status^Digital input 1;
                              .bLimitBackwardEnable := TIIB[SSL-EL7041]^STM Status^Status^Digital input 2;
                              .nRawEncoderULINT     := TIIB[IM1K3-EL5042]^FB Inputs Channel 1^Position'}
    M50: ST_MotionStage := (sName := 'QRIX:QUESTAR:MMS:02');
*)

END_VAR

// ---- POUs/PRG_1_PlcTask.TcPOU

PROGRAM PRG_1_PlcTask
VAR
END_VAR


PRG_2_PMPS();
PRG_3_LOG();
PRG_Diffractometer();
PRG_LAS();
PRG_SDS();
PRG_RotDet();
//PRG_Questar();
PRG_SpetrometerArm();
PRG_SSL();
PRG_Cryo();

END_PROGRAM

// ---- POUs/PRG_2_PMPS.TcPOU

PROGRAM PRG_2_PMPS
VAR
    fbArbiterIO: FB_SubSysToArbiter_IO;
END_VAR


GVL_PMPS.fbFastFaultOutput1.Execute();
GVL_PMPS.fbFastFaultOutput2.Execute();
fbArbiterIO(
    Arbiter:=GVL_PMPS.fbArbiter,
    fbFFHWO:=GVL_PMPS.fbFastFaultOutput1);

END_PROGRAM

// ---- POUs/PRG_3_LOG.TcPOU

PROGRAM PRG_3_LOG
VAR
      fbLogHandler: FB_LogHandler;
END_VAR


fbLogHandler();

END_PROGRAM

// ---- POUs/PRG_Diffractometer.TcPOU

PROGRAM PRG_Diffractometer
VAR
    fb_Diff_Theta : FB_MotionStage;
    fb_Diff_2Theta : FB_MotionStage;
    fb_Diff_2ThetaY : FB_MotionStage;
    fb_Diff_Chi : FB_MotionStage;
    fb_Diff_Phi : FB_MotionStage;
    fb_Diff_X : FB_MotionStage;
    fb_Diff_Y : FB_MotionStage;
    fb_Diff_Z : FB_MotionStage;
    bInit : BOOl := TRUE;

    //EPS
    EPS_Diff_Chi_Backward : FB_EPS;

    EPS_Diff_Phi_Forward : FB_EPS;

    EPS_Diff_Theta_Backward : FB_EPS;
    EPS_Diff_Theta_Forward : FB_EPS;

    EPS_Diff_X_Forward  : FB_EPS;
    EPS_Diff_X_Backward : FB_EPS;
    EPS_Diff_Y_Forward  : FB_EPS;
    EPS_Diff_Y_Backward : FB_EPS;
    EPS_Diff_Z_Forward  : FB_EPS;
    EPS_Diff_Z_Backward : FB_EPS;

    EPS_Diff_2Theta_Backward : FB_EPS;

    EPS_Diff_2ThetaY : FB_EPS;

    //Encoders for rotary stages
    fbSetPosition: MC_SetPosition;
    fb2ThetaAutoCoupling: FB_GantryAutoCoupling;
    couple : MC_GEARIN;
    decouple : MC_GEAROUT;
    bExecuteCouple: BOOL := TRUE;
    bExecuteDecouple: BOOL := FALSE;
    n2Theta AT %Q* :ULINT;
    r2Theta:LREAL;
    temp:ULINT;
    rtemp:LREAL;
    GantryDiff:REAL;

    fb_Diff_2Theta_Encoder : FB_MotionStage;

    eDiffXStateGet: E_DiffState;
    eDiffXStateSet: E_DiffState;
    astDiffXPosState: ARRAY[1..GeneralConstants.MAX_STATES] OF ST_PositionState;
    fbDiffXStage1D : FB_PositionState1D;

    eDiffYStateGet: E_DiffState;
    eDiffYStateSet: E_DiffState;
    astDiffYPosState: ARRAY[1..GeneralConstants.MAX_STATES] OF ST_PositionState;
    fbDiffYStage1D : FB_PositionState1D;

    eDiffZStateGet: E_DiffState;
    eDiffZStateSet: E_DiffState;
    astDiffZPosState: ARRAY[1..GeneralConstants.MAX_STATES] OF ST_PositionState;
    fbDiffZStage1D : FB_PositionState1D;

    eDiff2ThetaYStateGet: E_DiffState;
    eDiff2ThetaYStateSet: E_DiffState;
    astDiff2ThetaYPosState: ARRAY[1..GeneralConstants.MAX_STATES] OF ST_PositionState;
    fbDiff2ThetaYStage1D : FB_PositionState1D;

    eDiffPhiStateGet: E_DiffState;
    eDiffPhiStateSet: E_DiffState;
    astDiffPhiPosState: ARRAY[1..GeneralConstants.MAX_STATES] OF ST_PositionState;
    fbDiffPhiStage1D : FB_PositionState1D;

    eDiffChiStateGet: E_DiffState;
    eDiffChiStateSet: E_DiffState;
    astDiffChiPosState: ARRAY[1..GeneralConstants.MAX_STATES] OF ST_PositionState;
    fbDiffChiStage1D : FB_PositionState1D;

    eDiff2ThetaStateGet: E_DiffState;
    eDiff2ThetaStateSet: E_DiffState;
    astDiff2ThetaPosState: ARRAY[1..GeneralConstants.MAX_STATES] OF ST_PositionState;
    fbDiff2ThetaStage1D : FB_PositionState1D;

    eDiffThetaStateGet: E_DiffState;
    eDiffThetaStateSet: E_DiffState;
    astDiffThetaPosState: ARRAY[1..GeneralConstants.MAX_STATES] OF ST_PositionState;
    fbDiffThetaStage1D : FB_PositionState1D;

    fbStateSetup: FB_StateSetupHelper;
    stDefault: ST_PositionState := (
        fDelta := 0.5,
        fVelocity := 0.5,
        bMoveOk := TRUE,
        bValid := TRUE
    );
END_VAR


IF (bInit) THEN
    bInit := FALSE;
    Main.M28.bHardwareEnable := TRUE;
    Main.M28.bPowerSelf := TRUE;
    Main.M28.nBrakeMode := ENUM_StageBrakeMode.NO_BRAKE;
    Main.M28.nEnableMode := ENUM_StageEnableMode.DURING_MOTION;
    Main.M28.fVelocity := 0.1;

    Main.M29.bHardwareEnable := TRUE;
    Main.M29.bPowerSelf := TRUE;
    Main.M29.nBrakeMode := ENUM_StageBrakeMode.NO_BRAKE;
    Main.M29.nEnableMode := ENUM_StageEnableMode.DURING_MOTION;
    Main.M29.fVelocity := 0.1;

    Main.M30.bHardwareEnable := TRUE;
    Main.M30.bPowerSelf := TRUE;
    Main.M30.nBrakeMode := ENUM_StageBrakeMode.NO_BRAKE;
    Main.M30.nEnableMode := ENUM_StageEnableMode.DURING_MOTION;
    Main.M30.fVelocity := 0.1;

    Main.M31.bHardwareEnable := TRUE;
    Main.M31.bPowerSelf := TRUE;
    Main.M31.nBrakeMode := ENUM_StageBrakeMode.NO_BRAKE;
    Main.M31.nEnableMode := ENUM_StageEnableMode.DURING_MOTION;
    Main.M31.fVelocity := 0.1;

    Main.M32.bHardwareEnable := TRUE;
    Main.M32.bPowerSelf := TRUE;
    Main.M32.nBrakeMode := ENUM_StageBrakeMode.NO_BRAKE;
    Main.M32.nEnableMode := ENUM_StageEnableMode.DURING_MOTION;
    Main.M32.fVelocity := 0.1;

    Main.M33.bHardwareEnable := TRUE;
    Main.M33.bPowerSelf := TRUE;
    Main.M33.nBrakeMode := ENUM_StageBrakeMode.NO_BRAKE;
    Main.M33.nEnableMode := ENUM_StageEnableMode.DURING_MOTION;
    Main.M33.fVelocity := 0.1;

    Main.M34.bHardwareEnable := TRUE;
    Main.M34.bPowerSelf := TRUE;
    Main.M34.nBrakeMode := ENUM_StageBrakeMode.NO_BRAKE;
    Main.M34.nEnableMode := ENUM_StageEnableMode.DURING_MOTION;
    Main.M34.fVelocity := 0.1;

    Main.M35.bHardwareEnable := TRUE;
    Main.M35.bPowerSelf := TRUE;
    Main.M35.nBrakeMode := ENUM_StageBrakeMode.NO_BRAKE;
    Main.M35.nEnableMode := ENUM_StageEnableMode.DURING_MOTION;
    Main.M35.fVelocity := 0.1;

    fbStateSetup(stPositionState:=stDefault, bSetDefault:=TRUE);

    fbStateSetup(stPositionState:=astDiffXPosState[E_DiffState.TRANSFER_ARM_INTERFACE], sName:='TRANSFER_ARM_INTERFACE',
        fPosition := 0
    );
    fbStateSetup(stPositionState:=astDiffYPosState[E_DiffState.TRANSFER_ARM_INTERFACE], sName:='TRANSFER_ARM_INTERFACE',
        fPosition := 0
    );
    fbStateSetup(stPositionState:=astDiffZPosState[E_DiffState.TRANSFER_ARM_INTERFACE], sName:='TRANSFER_ARM_INTERFACE',
        fPosition := 0
    );
    fbStateSetup(stPositionState:=astDiff2ThetaYPosState[E_DiffState.TRANSFER_ARM_INTERFACE], sName:='TRANSFER_ARM_INTERFACE',
        fPosition := 0
    );
    fbStateSetup(stPositionState:=astDiffPhiPosState[E_DiffState.TRANSFER_ARM_INTERFACE], sName:='TRANSFER_ARM_INTERFACE',
        fPosition := 0
    );
    fbStateSetup(stPositionState:=astDiffChiPosState[E_DiffState.TRANSFER_ARM_INTERFACE], sName:='TRANSFER_ARM_INTERFACE',
        fPosition := 0
    );
    fbStateSetup(stPositionState:=astDiff2ThetaPosState[E_DiffState.TRANSFER_ARM_INTERFACE], sName:='TRANSFER_ARM_INTERFACE',
        fPosition := 0
    );
    fbStateSetup(stPositionState:=astDiffThetaPosState[E_DiffState.TRANSFER_ARM_INTERFACE], sName:='TRANSFER_ARM_INTERFACE',
        fPosition := 0
    );


    fbStateSetup(stPositionState:=astDiffXPosState[E_DiffState.NOMINAL_POSITION], sName:='NOMINAL_POSITION',
        fPosition := 0
    );
    fbStateSetup(stPositionState:=astDiffYPosState[E_DiffState.NOMINAL_POSITION], sName:='NOMINAL_POSITION',
        fPosition := 0
    );
    fbStateSetup(stPositionState:=astDiffZPosState[E_DiffState.NOMINAL_POSITION], sName:='NOMINAL_POSITION',
        fPosition := 0
    );
    fbStateSetup(stPositionState:=astDiff2ThetaYPosState[E_DiffState.NOMINAL_POSITION], sName:='NOMINAL_POSITION',
        fPosition := 0
    );
    fbStateSetup(stPositionState:=astDiffPhiPosState[E_DiffState.NOMINAL_POSITION], sName:='NOMINAL_POSITION',
        fPosition := 0
    );
    fbStateSetup(stPositionState:=astDiffChiPosState[E_DiffState.NOMINAL_POSITION], sName:='NOMINAL_POSITION',
        fPosition := 0
    );
    fbStateSetup(stPositionState:=astDiff2ThetaPosState[E_DiffState.NOMINAL_POSITION], sName:='NOMINAL_POSITION',
        fPosition := 0
    );
    fbStateSetup(stPositionState:=astDiffThetaPosState[E_DiffState.NOMINAL_POSITION], sName:='NOMINAL_POSITION',
        fPosition := 0
    );
END_IF

//EPS

// All bits must be TRUE to enable the specified direction (backward or forward)
// The bits are populated right to left in typhos screen. So Descriptions highest bit number is at the beginning of the description.
// The eps IN_OUT variable must be assigned before using the FB_EPS in any way.

// DIFFRACTOMETER THETA ANGLE RESTRICTIONS
// Disable movement in negative direction.
EPS_Diff_Theta_Backward(eps:=Main.M34.stEPSBackwardEnable);
EPS_Diff_Theta_Backward.setDescription('NEGATIVE MOTION'); // SET DESCRIPTION FOR BYTE INDICATOR LABELS
EPS_Diff_Theta_Backward.setBit(nBits:= 3,
    bValue := Main.M34.Axis.NcToPlc.ActPos - Main.M49.Axis.NcToPlc.ActPos > -1.0
);
// Diffractometer Theta cannot go less than 5 degrees if the Diffractometer Chi is less than -5 degrees
EPS_Diff_Theta_Backward.setBit(nBits:= 2, bValue:=F_CheckAxisGEQ(Main.M34,5) OR F_CheckAxisGEQ(Main.M33,-5));
// Diffractometer Theta cannot go less than 10 degrees if the MID IR (LAS VIS) is IN, which is defined as a position of 90 +/- 1.
EPS_Diff_Theta_Backward.setBit(nBits:= 1, bValue:= F_CheckAxisGRT(Main.M34,10) OR F_Limit(Main.M36.stAxisStatus.fActPosition, 91, 89, false));
// Diffractometer Theta cannot go less than 10 degrees if the Diffractometer phi is at 90 +/- 1.
EPS_Diff_Theta_Backward.setBit(nBits:= 0, bValue:=F_CheckAxisGRT(Main.M34,10) OR F_Limit(Main.M32.stAxisStatus.fActPosition, 91, 89, false));

// Disable movement in positive direction.
EPS_Diff_Theta_Forward(eps:=Main.M34.stEPSForwardEnable);
EPS_Diff_Theta_Forward.setDescription('POSITIVE MOTION'); // SET DESCRIPTION FOR BYTE INDICATOR LABELS
EPS_Diff_Theta_Forward.setBit(nBits:= 1,
    bValue := Main.M34.Axis.NcToPlc.ActPos - Main.M49.Axis.NcToPlc.ActPos < 1.0
);
// Diffractometer Theta cannot go more than Diffractometer 2Theta plus 21 degrees
EPS_Diff_Theta_Forward.setBit(nBits:= 0, bValue:=Main.M34.Axis.NcToPlc.ActPos < Main.M35.stAxisStatus.fActPosition+21);

// DIFFRACTOMETER CHI ANGLE RESTRICTIONS
// Disable movement in negative direction.
EPS_Diff_Chi_Backward(eps:=Main.M33.stEPSBackwardEnable);
EPS_Diff_Chi_Backward.setDescription('NEGATIVE MOTION'); // SET DESCRIPTION FOR BYTE INDICATOR LABELS
// Diffractometer Chi cannot go less than -5 degrees if the Diffractometer Theta is less than 5 degrees
EPS_Diff_Chi_Backward.setBit(nBits:= 0, bValue:=F_CheckAxisGEQ(Main.M33,-5) OR F_CheckAxisGEQ(Main.M34,5));

// DIFFRACTOMETER PHI ANGLE RESTRICTIONS
// Disable movement in positive direction.
EPS_Diff_Phi_Forward(eps:=Main.M32.stEPSForwardEnable);
EPS_Diff_Phi_Forward.setDescription('POSITIVE MOTION'); // SET DESCRIPTION FOR BYTE INDICATOR LABELS
// Diffractometer Phi cannot go greater than 45 degrees when the MID IR (LAS VIS) is greater than 45 degrees
EPS_Diff_Phi_Forward.setBit(nBits:= 1, bValue:=Main.M36.Axis.NcToPlc.ActPos <= 45 OR Main.M32.Axis.NcToPlc.ActPos <= 5);
// Diffractometer Phi cannot go greater than 45 degrees when theta is within 1 degree of 0 degrees.
EPS_Diff_Phi_Forward.setBit(nBits:= 0, bValue:=Main.M32.Axis.NcToPlc.ActPos <= 45 OR F_Limit(Main.M34.stAxisStatus.fActPosition, 1, -1, false));

// DIFFRACTOMETER Z POSITION RESTRICTIONS
// Disable movement in negative direction.
EPS_Diff_Z_Backward(eps:=Main.M30.stEPSBackwardEnable);
EPS_Diff_Z_Backward.setDescription('NEGATIVE MOTION'); // SET DESCRIPTION FOR BYTE INDICATOR LABELS
EPS_Diff_Z_Backward.setBit(nBits:= 1,
    bValue := Main.M30.Axis.NcToPlc.ActPos - (Main.M48.Axis.NcToPlc.ActPos - GVL_VAR.fCryoZNeutralPositionAtDiffZ0) > -1.0
);
// Diffractometer Z cannot go less than 5mm when the diagonal paddle horizontal (LAS_D_H) position is greater than 50 mm.
EPS_Diff_Z_Backward.setBit(nBits:= 0, bValue:=Main.M37.Axis.NcToPlc.ActPos <= 50 OR Main.M30.Axis.NcToPlc.ActPos >= 5);

// Disable movement in positive direction
EPS_Diff_Z_Forward(eps:=Main.M30.stEPSForwardEnable);
EPS_Diff_Z_Forward.setDescription('POSITIVE MOTION'); // SET DESCRIPTION FOR BYTE INDICATOR LABELS
EPS_Diff_Z_Forward.setBit(nBits:= 0,
    bValue := Main.M30.Axis.NcToPlc.ActPos - (Main.M48.Axis.NcToPlc.ActPos - GVL_VAR.fCryoZNeutralPositionAtDiffZ0) < 1.0
);

// Diff X
// Disable movement in negative direction.
EPS_Diff_X_Backward(eps:=Main.M28.stEPSBackwardEnable);
EPS_Diff_X_Backward.setDescription('NEGATIVE MOTION'); // SET DESCRIPTION FOR BYTE INDICATOR LABELS
EPS_Diff_X_Backward.setBit(nBits:= 0,
    bValue := Main.M28.Axis.NcToPlc.ActPos - Main.M46.Axis.NcToPlc.ActPos > -1.0
);

// Disable movement in positive direction
EPS_Diff_X_Forward(eps:=Main.M28.stEPSForwardEnable);
EPS_Diff_X_Forward.setDescription('POSITIVE MOTION'); // SET DESCRIPTION FOR BYTE INDICATOR LABELS
EPS_Diff_X_Forward.setBit(nBits:= 0,
    bValue := Main.M28.Axis.NcToPlc.ActPos - Main.M46.Axis.NcToPlc.ActPos < 1.0
);

// Diff Y
// Disable movement in negative direction.
EPS_Diff_Y_Backward(eps:=Main.M29.stEPSBackwardEnable);
EPS_Diff_Y_Backward.setDescription('NEGATIVE MOTION'); // SET DESCRIPTION FOR BYTE INDICATOR LABELS
EPS_Diff_Y_Backward.setBit(nBits:= 0,
    bValue := Main.M47.Axis.NcToPlc.ActPos - F_TargetCryoYPosition(
        fNeutralPosition := GVL_VAR.fCryoYNeutralPositionAtDiffY0 + Main.M29.Axis.NcToPlc.ActPos,
        fBraidDiameter   := GVL_VAR.fBraidDiameter,
        fPhiAngleDeg     := Main.M32.Axis.NcToPlc.ActPos) < 1.0
);

// Disable movement in positive direction
EPS_Diff_Y_Forward(eps:=Main.M29.stEPSForwardEnable);
EPS_Diff_Y_Forward.setDescription('POSITIVE MOTION'); // SET DESCRIPTION FOR BYTE INDICATOR LABELS
EPS_Diff_Y_Forward.setBit(nBits:= 0,
    bValue := Main.M47.Axis.NcToPlc.ActPos - F_TargetCryoYPosition(
        fNeutralPosition := GVL_VAR.fCryoYNeutralPositionAtDiffY0 + Main.M29.Axis.NcToPlc.ActPos,
        fBraidDiameter   := GVL_VAR.fBraidDiameter,
        fPhiAngleDeg     := Main.M32.Axis.NcToPlc.ActPos) > -1.0
);

// DIFFRACTOMETER 2-THETA ANGLE RESTRICTIONS
// Disable movement in negative direction.
EPS_Diff_2Theta_Backward(eps:=Main.M35.stEPSBackwardEnable);
EPS_Diff_2Theta_Backward.setDescription('NEGATIVE MOTION'); // SET DESCRIPTION FOR BYTE INDICATOR LABELS
// Diffractometer 2 Theta cannot go less than the diffractometer theta angle minus 21 degrees.
EPS_Diff_2Theta_Backward.setBit(nBits:= 0, bValue:=Main.M35.Axis.NcToPlc.ActPos > Main.M34.stAxisStatus.fActPosition - 21);

fb_Diff_X(stMotionStage:=Main.M28);
fb_Diff_Y(stMotionStage:=Main.M29);
fb_Diff_Z(stMotionStage:=Main.M30);
fb_Diff_2ThetaY(stMotionStage:=Main.M31);
fb_Diff_Phi(stMotionStage:=Main.M32);
fb_Diff_Chi(stMotionStage:=Main.M33);
fb_Diff_Theta(stMotionStage:=Main.M34);
fb_Diff_2Theta(stMotionStage:=Main.M35);

END_PROGRAM

// ---- POUs/F_CheckAxisGEQ.TcPOU

FUNCTION F_CheckAxisGEQ : BOOL
VAR_INPUT
    stMotionStage: ST_MotionStage;
    fQueryValue: LREAL;
END_VAR
VAR
END_VAR


F_CheckAxisGEQ := F_CheckAxis(stMotionStage, 3, fQueryValue);

END_FUNCTION

// ---- POUs/F_CheckAxis.TcPOU

FUNCTION F_CheckAxis : BOOL
VAR_INPUT
    stMotionStage: ST_MotionStage;
    nComparisonCode: UINT;
    fQueryValue: LREAL;
END_VAR
VAR
END_VAR


CASE nComparisonCode OF
    0: F_CheckAxis := stMotionStage.stAxisStatus.fActPosition <  fQueryValue AND stMotionStage.fPosition <  fQueryValue; // <
    1: F_CheckAxis := stMotionStage.stAxisStatus.fActPosition <= fQueryValue AND stMotionStage.fPosition <= fQueryValue; // <=
    2: F_CheckAxis := stMotionStage.stAxisStatus.fActPosition >  fQueryValue AND stMotionStage.fPosition >  fQueryValue; // >
    3: F_CheckAxis := stMotionStage.stAxisStatus.fActPosition >= fQueryValue AND stMotionStage.fPosition >= fQueryValue; // <=
ELSE
    return;
END_CASE;

END_FUNCTION

// ---- POUs/F_CheckAxisGRT.TcPOU

FUNCTION F_CheckAxisGRT : BOOL
VAR_INPUT
    stMotionStage: ST_MotionStage;
    fQueryValue: LREAL;
END_VAR
VAR
END_VAR


F_CheckAxisGRT := F_CheckAxis(stMotionStage, 2, fQueryValue);

END_FUNCTION

// ---- POUs/F_Limit.TcPOU

FUNCTION F_Limit : BOOL
VAR_INPUT
    fVal : LREAL;
    fLLim : LREAL;
    fHLim : LREAL;
    bInclusive : BOOL;
END_VAR
VAR
END_VAR


IF bInclusive THEN
    IF fLLim <= fHLim THEN
        F_Limit := fLLim <= fVal AND fHLim >= fVal;
    ELSE
        F_Limit := fLLim >= fVal OR fHLim <= fVal;
    END_IF
ELSE
    IF fLLim <= fHLim THEN
        F_Limit := fLLim < fVal AND fHLim > fVal;
    ELSE
        F_Limit := fLLim > fVal OR fHLim < fVal;
    END_IF
END_IF

END_FUNCTION

// ---- POUs/F_TargetCryoYPosition.TcPOU

FUNCTION F_TargetCryoYPosition : LREAL
VAR_INPUT
    fNeutralPosition : LREAL;
    fBraidDiameter   : LREAL;
    fPhiAngleDeg     : LREAL;
END_VAR


F_TargetCryoYPosition := fNeutralPosition - ABS(fBraidDiameter * (1 - Cos(fPhiAngleDeg * 3.1415 / 180)));

END_FUNCTION

// ---- POUs/PRG_LAS.TcPOU

PROGRAM PRG_LAS
VAR
    fb_LAS_VIS : FB_MotionStage;
    fb_LAS_D_H : FB_MotionStage;
    fb_LAS_D_V : FB_MotionStage;
    bInit : BOOl := TRUE;

    //LAS_VIS BEAM OK/NOK
    {attribute 'pytmc' := '
      pv: QRIX:LAS:MMS:VIS:STATES:SET
      io: io
    '}
    eLAS_VIS_StateSet: ENUM_LAS_VIS_States;
    {attribute 'pytmc' := '
      pv: QRIX:LAS:MMS:VIS:STATES:GET
      io: i
    '}
    eLAS_VIS_StateGet: ENUM_LAS_VIS_States;
    {attribute 'pytmc' := 'pv: QRIX:LAS:MMS:VIS'}
    fbLAS_VIS_PositionState1D : FB_PositionState1D;
    astLAS_VIS_PositionState : ARRAY [1..GeneralConstants.MAX_STATES] of ST_PositionState;
    fbLAS_VIS_StateSetupHelper : FB_StateSetupHelper;
    fbLAS_VIS_HardwareFFOutput : FB_HardwareFFOutput;

    //EPS
    stLAS_VIS : DUT_EPS;
    fbLAS_VIS_EPS : FB_EPS;

    stLAS_D_H : DUT_EPS;
    fbLAS_D_H_EPS : FB_EPS;
END_VAR


IF (bInit) THEN
    bInit := FALSE;
    Main.M36.bHardwareEnable := TRUE;
    Main.M36.bPowerSelf := TRUE;
    Main.M36.nBrakeMode := ENUM_StageBrakeMode.NO_BRAKE;
    Main.M36.nEnableMode := ENUM_StageEnableMode.DURING_MOTION;
    Main.M36.fVelocity := 0.1;

    Main.M37.bHardwareEnable := TRUE;
    Main.M37.bPowerSelf := TRUE;
    Main.M37.nBrakeMode := ENUM_StageBrakeMode.NO_BRAKE;
    Main.M37.nEnableMode := ENUM_StageEnableMode.DURING_MOTION;
    Main.M37.fVelocity := 0.1;

    Main.M38.bHardwareEnable := TRUE;
    Main.M38.bPowerSelf := TRUE;
    Main.M38.nBrakeMode := ENUM_StageBrakeMode.NO_BRAKE;
    Main.M38.nEnableMode := ENUM_StageEnableMode.DURING_MOTION;
    Main.M38.fVelocity := 0.1;

    // Initialize the M36 LAS VIS Axis States
    // Beam OK if one of these two states is active. Otherwise, beam is not okay.
    fbLAS_VIS_StateSetupHelper(stPositionState := astLAS_VIS_PositionState[1], sName := 'Position7to24mm', bValid := TRUE, fPosition := 15.5, fDelta := 8.5);
    fbLAS_VIS_StateSetupHelper(stPositionState := astLAS_VIS_PositionState[2], sName := 'Position62to77mm', bValid := TRUE, fPosition := 69.5, fDelta := 7.5);

END_IF
//EPS
(*
fbLAS_D_H_EPS.setDescription('Less10mm;SampleZ;PHI'); // SET DESCRITION FOR BYTE INDICATOR LABELS
//Zero is fully retracted
fbLAS_D_H_EPS.setBit(nBits:= 0, bValue:=fb_LAS_D_H.stMotionStage.fPosition<=10);
fbLAS_D_H_EPS.setBit(nBits:= 1, bValue:=fb_LAS_D_H.stMotionStage.fPosition<=10 OR PRG_Diffractometer.fb_Diff_Z.stMotionStage.fPosition<=-20);
fbLAS_D_H_EPS.setBit(nBits:= 2, bValue:=fb_LAS_D_H.stMotionStage.fPosition<=10 OR PRG_Diffractometer.fb_Diff_Phi.stMotionStage.fPosition>0);
fbLAS_D_H_EPS(eps:=stLAS_D_H);
fb_LAS_D_H.stMotionStage.stEPSForwardEnable := stLAS_D_H; // Update Motion stage structure.

fbLAS_VIS_EPS.setDescription('IN90mm;PHIat90;Theta<10'); // SET DESCRITION FOR BYTE INDICATOR LABELS
//Zero is fully retracted
fbLAS_VIS_EPS.setBit(nBits:= 0, bValue:=fb_LAS_VIS.stMotionStage.fPosition<=5);
fbLAS_VIS_EPS.setBit(nBits:= 1, bValue:=fb_LAS_VIS.stMotionStage.fPosition<=5 OR PRG_Diffractometer.fb_Diff_Phi.stMotionStage.fPosition<>90);
fbLAS_VIS_EPS.setBit(nBits:= 2, bValue:=fb_LAS_VIS.stMotionStage.fPosition<=5 OR PRG_Diffractometer.fb_Diff_Theta.stMotionStage.fPosition>10);
fbLAS_VIS_EPS(eps:=fbLAS_VIS_EPS);
//fb_LAS_VIS.stMotionStage.stEPSForwardEnable := fbLAS_VIS_EPS;
*)

fbLAS_VIS_PositionState1D(
    stMotionStage := Main.M36,
    astPositionState := astLAS_VIS_PositionState,
    eEnumSet := eLAS_VIS_StateSet,
    eEnumGet := eLAS_VIS_StateGet,
    bEnable := TRUE
);

IF eLAS_VIS_StateGet = ENUM_LAS_VIS_States.Position7to24mm OR eLAS_VIS_StateGet = ENUM_LAS_VIS_States.Position62to77mm THEN
    // BEAM OKAY

ELSE
    // BEAM NOT OKAY
END_IF

fb_LAS_VIS(stMotionStage:=Main.M36);
fb_LAS_D_H(stMotionStage:=Main.M37);
fb_LAS_D_V(stMotionStage:=Main.M38);

END_PROGRAM

// ---- POUs/PRG_SDS.TcPOU

PROGRAM PRG_SDS
VAR
    fb_SDS_ROT_V : FB_MotionStage;
    fb_SDS_X : FB_MotionStage;
    fb_SDS_Y : FB_MotionStage;
    fb_SDS_Z : FB_MotionStage;
    fb_SDS_ROT_H : FB_MotionStage;
    fb_SDS_H : FB_MotionStage;
    bInit : BOOl := TRUE;

    EPS_SDS_H_Backward : FB_EPS;
    EPS_SDS_H_Forward : FB_EPS;
    fSDSYEPSOverride: REAL;

    EPS_SDS_Y_Backward : FB_EPS;
    EPS_SDS_Y_Forward : FB_EPS;

    fMaxSampleDeliveryArmPositionWithValveClosed : REAL := 50;

    {attribute 'pytmc' := '
        pv: QRIX:SDS:NP
        field: DESC Structure defining qrixs sample delivery system non-persistent data.
    '}
    stSDS: ST_SDS;
    fbSDS: FB_SDS;

    {attribute 'pytmc' := '
        pv: QRIX:SDS:Y:EPS:BACK:OVRD
        field: DESC Allow SDS Y backward limit to be user defined for 1h.
    '}
    bEPS_SDS_Y_Backward_Override : BOOL;
    fbEPS_SDS_Y_Backward_Override_Start : R_TRIG;
    tEPS_SDS_Y_Backward_Override_Time : TIME := T#1h;
    fbEPS_SDS_Y_EPS_BACK_OVRD_TIMER : TON;

    {attribute 'pytmc' := '
        pv: QRIX:SDS:Y:EPS:BACK:OVRD_COUNTDOWN
        field: DESC Time Remaining Untill Override resets.
    '}
    tSDS_Y_EPS_BACK_OVRD_TimerCountDown : STRING := TIME_TO_STRING(T#0s);

    {attribute 'pytmc' := '
        pv: QRIX:SDS:Y:EPS:BACK:USR:OVRD_LIM
        field: DESC Allow SDS Y backward limit to be user defined for 1h.
        io: io
        autosave_pass1: VAL DESC
    '}
    fSDS_Y_NEGATIVE_LIM_USR : LREAL;
    {attribute 'pytmc' := '
        pv: QRIX:SDS:Y:EPS:BACK:OVRD_LIM
        field: DESC Readback from Actual Soft Limit.
        io: i
    '}
    fSDS_Y_NEGATIVE_LIM : LREAL;
    fSDS_Y_NEGATIVE_LIM_DEFAULT  : LREAL := -110;


END_VAR
VAR PERSISTENT
    {attribute 'pytmc' := '
        pv: QRIX:SDS:P
        field: DESC Structure defining qrixs sample delivery system persistent data.
    '}
    stSDSPersistent: ST_SDSPersistent;
END_VAR


IF bInit THEN
    bInit := FALSE;
    Main.M39.bHardwareEnable := TRUE;
    Main.M39.bPowerSelf := TRUE;
    Main.M39.nBrakeMode := ENUM_StageBrakeMode.NO_BRAKE;
    Main.M39.nEnableMode := ENUM_StageEnableMode.DURING_MOTION;

    Main.M40.bHardwareEnable := TRUE;
    Main.M40.bPowerSelf := TRUE;
    Main.M40.nBrakeMode := ENUM_StageBrakeMode.NO_BRAKE;
    Main.M40.nEnableMode := ENUM_StageEnableMode.DURING_MOTION;

    Main.M41.bHardwareEnable := TRUE;
    Main.M41.bPowerSelf := TRUE;
    Main.M41.nBrakeMode := ENUM_StageBrakeMode.NO_BRAKE;
    Main.M41.nEnableMode := ENUM_StageEnableMode.DURING_MOTION;

    Main.M42.bHardwareEnable := TRUE;
    Main.M42.bPowerSelf := TRUE;
    Main.M42.nBrakeMode := ENUM_StageBrakeMode.NO_BRAKE;
    Main.M42.nEnableMode := ENUM_StageEnableMode.DURING_MOTION;
    Main.M42.nHomingMode := ENUM_EpicsHomeCmd.HOME_VIA_LOW;
    Main.M42.bLimitBackwardEnable := TRUE;
    Main.M42.bLimitForwardEnable := TRUE;

    Main.M43.bHardwareEnable := TRUE;
    Main.M43.bPowerSelf := TRUE;
    Main.M43.nBrakeMode := ENUM_StageBrakeMode.NO_BRAKE;
    Main.M43.nEnableMode := ENUM_StageEnableMode.DURING_MOTION;
    Main.M43.nHomingMode := ENUM_EpicsHomeCmd.LOW_LIMIT;
    Main.M43.fHomePosition := 0.0;

    Main.M44.bHardwareEnable := TRUE;
    Main.M44.bPowerSelf := TRUE;
    Main.M44.nBrakeMode := ENUM_StageBrakeMode.NO_BRAKE;
    Main.M44.nEnableMode := ENUM_StageEnableMode.DURING_MOTION;
    Main.M44.nHomingMode := ENUM_EpicsHomeCmd.HOME_VIA_LOW;
    Main.M44.fHomePosition := 0;//1.176; distance from home switch trigger to lower limit trigger

    fSDSYEPSOverride := -40;
    fSDS_Y_NEGATIVE_LIM := fSDS_Y_NEGATIVE_LIM_DEFAULT;
END_IF

GVL_Interface.QRIX_MOT_SDS_MMS_H_RAW_ENC_CNTS := Main.M44.nRawEncoderUINT;
GVL_Interface.QRIX_MOT_SDS_MMS_H_FORWARD_EN := Main.M44.bLimitForwardEnable;
GVL_Interface.QRIX_MOT_SDS_MMS_H_BACKWARD_EN := Main.M44.bLimitBackwardEnable;

//EPS

// Sample Delivery System
// Disable movement in negative direction.
EPS_SDS_H_Backward(eps:=Main.M44.stEPSBackwardEnable);
EPS_SDS_H_Backward.setDescription('NEGATIVE MOTION ALLOWED UNTIL LIMIT'); // SET DESCRIPTION FOR BYTE INDICATOR LABELS

// Disable movement in positive direction.
EPS_SDS_H_Forward(eps:=Main.M44.stEPSForwardEnable);
EPS_SDS_H_Forward.setDescription('POS MOTION IF VGC_03 closed: (cmd<50mm | pos<50mm | Homing Valid | SDS Y<-45mm)'); // SET DESCRIPTION FOR BYTE INDICATOR LABELS
// Sample Delivery Arm can Extend if the VGC valve is open and not closed, and it has been homed.
EPS_SDS_H_Forward.setBit(nBits:= 4, bValue:= NOT stSDS.tonForwardHomingLimit.Q);
EPS_SDS_H_Forward.setBit(nBits:= 3, bValue:=(NOT GVL_Interface.QRIX_VAC_VGC_03_CLOSED_LIMIT_SWITCH AND
    GVL_Interface.QRIX_VAC_VGC_03_OPEN_LIMIT_SWITCH) OR Main.M44.stAxisStatus.fPosition < fMaxSampleDeliveryArmPositionWithValveClosed);
EPS_SDS_H_Forward.setBit(nBits:= 2, bValue:=(NOT GVL_Interface.QRIX_VAC_VGC_03_CLOSED_LIMIT_SWITCH AND
    GVL_Interface.QRIX_VAC_VGC_03_OPEN_LIMIT_SWITCH) OR Main.M44.stAxisStatus.fActPosition < fMaxSampleDeliveryArmPositionWithValveClosed);
EPS_SDS_H_Forward.setBit(nBits:= 1, bValue:=(NOT GVL_Interface.QRIX_VAC_VGC_03_CLOSED_LIMIT_SWITCH AND
    GVL_Interface.QRIX_VAC_VGC_03_OPEN_LIMIT_SWITCH) OR NOT stSDS.bHomingRequired);
EPS_SDS_H_Forward.setBit(nBits:= 0, bValue:=(NOT GVL_Interface.QRIX_VAC_VGC_03_CLOSED_LIMIT_SWITCH AND
    GVL_Interface.QRIX_VAC_VGC_03_OPEN_LIMIT_SWITCH) OR Main.M40.stAxisStatus.fActPosition < fSDSYEPSOverride);


// Disable movement in negative direction.
EPS_SDS_Y_Backward(eps:=Main.M40.stEPSBackwardEnable);
EPS_SDS_Y_Backward.setDescription('NEGATIVE MOTION ALLOWED UNTIL LIMIT'); // SET DESCRIPTION FOR BYTE INDICATOR LABELS

EPS_SDS_Y_Backward.setBit(nBits:=0, bValue:= Main.M40.stAxisStatus.fActPosition > fSDS_Y_NEGATIVE_LIM);

fbEPS_SDS_Y_EPS_BACK_OVRD_TIMER(IN:=bEPS_SDS_Y_Backward_Override, PT:= tEPS_SDS_Y_Backward_Override_Time);
tSDS_Y_EPS_BACK_OVRD_TimerCountDown := TIME_TO_STRING(tEPS_SDS_Y_Backward_Override_Time - fbEPS_SDS_Y_EPS_BACK_OVRD_TIMER.ET);

IF bEPS_SDS_Y_Backward_Override THEN
    fSDS_Y_NEGATIVE_LIM := fSDS_Y_NEGATIVE_LIM_USR;
END_IF

// Resets timer when EPS timer has expired; 1hr default
IF fbEPS_SDS_Y_EPS_BACK_OVRD_TIMER.Q THEN
    bEPS_SDS_Y_Backward_Override := FALSE;
    fSDS_Y_NEGATIVE_LIM := fSDS_Y_NEGATIVE_LIM_DEFAULT;
END_IF



// Disable movement in positive direction.
EPS_SDS_Y_Forward(eps:=Main.M40.stEPSForwardEnable);
EPS_SDS_Y_Forward.setDescription('POSITIVE MOTION ALLOWED UNTIL LIMIT'); // SET DESCRIPTION FOR BYTE INDICATOR LABELS

fb_SDS_X(stMotionStage:=Main.M39);
fb_SDS_Y(stMotionStage:=Main.M40);
fb_SDS_Z(stMotionStage:=Main.M41);

Main.M42.bHome := NOT Main.M42.bHome;

fb_SDS_ROT_V(stMotionStage:=Main.M42);
fb_SDS_ROT_H(stMotionStage:=Main.M43);
fb_SDS_H(stMotionStage:=Main.M44);

stSDS.stGarageYStage REF= Main.M40;
stSDS.stGarageRStage REF= Main.M42;
stSDS.stTransferArmHStage REF= Main.M44;
stSDS.stTransferArmRStage REF= Main.M43;

stSDS.eDiffXStateGet REF= PRG_Diffractometer.eDiffXStateGet;
stSDS.eDiffXStateSet REF= PRG_Diffractometer.eDiffXStateSet;
stSDS.stDiffXStage REF= Main.M28;

stSDS.eDiffYStateGet REF= PRG_Diffractometer.eDiffYStateGet;
stSDS.eDiffYStateSet REF= PRG_Diffractometer.eDiffYStateSet;
stSDS.stDiffYStage REF= Main.M29;

stSDS.eDiffZStateGet REF= PRG_Diffractometer.eDiffZStateGet;
stSDS.eDiffZStateSet REF= PRG_Diffractometer.eDiffZStateSet;
stSDS.stDiffZStage REF= Main.M30;

stSDS.eDiff2ThetaYStateGet REF= PRG_Diffractometer.eDiff2ThetaYStateGet;
stSDS.eDiff2ThetaYStateSet REF= PRG_Diffractometer.eDiff2ThetaYStateSet;
stSDS.stDiff2ThetaYStage REF= Main.M31;

stSDS.eDiffPhiStateGet REF= PRG_Diffractometer.eDiffPhiStateGet;
stSDS.eDiffPhiStateSet REF= PRG_Diffractometer.eDiffPhiStateSet;
stSDS.stDiffPhiStage REF= Main.M32;

stSDS.eDiffChiStateGet REF= PRG_Diffractometer.eDiffChiStateGet;
stSDS.eDiffChiStateSet REF= PRG_Diffractometer.eDiffChiStateSet;
stSDS.stDiffChiStage REF= Main.M33;

stSDS.eDiff2ThetaStateGet REF= PRG_Diffractometer.eDiff2ThetaStateGet;
stSDS.eDiff2ThetaStateSet REF= PRG_Diffractometer.eDiff2ThetaStateSet;
stSDS.stDiff2ThetaStage REF= Main.M34;

stSDS.eDiffThetaStateGet REF= PRG_Diffractometer.eDiffThetaStateGet;
stSDS.eDiffThetaStateSet REF= PRG_Diffractometer.eDiffThetaStateSet;
stSDS.stDiffThetaStage REF= Main.M35;

// Function block containing logic for sample delivery system motion automation.
fbSDS(
    stSDSin := stSDS,
    stSDSPersistent := stSDSPersistent
);

END_PROGRAM

// ---- Devices/FB_SDS.TcPOU

FUNCTION_BLOCK FB_SDS
VAR_IN_OUT
    stSDSin : ST_SDS;
    stSDSPersistent : ST_SDSPersistent;
END_VAR
VAR
    nIndex: UINT;

    fbStateSetup: FB_StateSetupHelper;
    stDefault: ST_PositionState := (
        fDelta := 0.5,
        fVelocity := 1,
        bMoveOk := TRUE,
        bValid := TRUE
    );
END_VAR


// Check the present homing status
ACT_CheckHomeStatus();

IF NOT stSDSPersistent.bInitialized THEN
    // Do all the required initialization for the persistent data of the sample delivery system.

    stSDSPersistent.stTransferArmSlot.sTag := 'TA';
    stSDSPersistent.stDiffractometerSlot.sTag := 'DF';

    FOR nIndex := E_SDSGarageYStates.T1 to E_SDSGarageYStates.B4 BY 1 DO
        stSDSPersistent.astGarageSlot[nIndex].eState := E_SampleSlotStates.EMPTY;
        stSDSPersistent.astGarageSlot[nIndex].sDesc  := '';
    END_FOR

    stSDSPersistent.astGarageSlot[E_SDSGarageYStates.T1].sTag := 'T1';
    stSDSPersistent.astGarageSlot[E_SDSGarageYStates.T2].sTag := 'T2';
    stSDSPersistent.astGarageSlot[E_SDSGarageYStates.T3].sTag := 'T3';
    stSDSPersistent.astGarageSlot[E_SDSGarageYStates.T4].sTag := 'T4';
    stSDSPersistent.astGarageSlot[E_SDSGarageYStates.M1].sTag := 'M1';
    stSDSPersistent.astGarageSlot[E_SDSGarageYStates.M2].sTag := 'M2';
    stSDSPersistent.astGarageSlot[E_SDSGarageYStates.M3].sTag := 'M3';
    stSDSPersistent.astGarageSlot[E_SDSGarageYStates.M4].sTag := 'M4';
    stSDSPersistent.astGarageSlot[E_SDSGarageYStates.B1].sTag := 'B1';
    stSDSPersistent.astGarageSlot[E_SDSGarageYStates.B2].sTag := 'B2';
    stSDSPersistent.astGarageSlot[E_SDSGarageYStates.B3].sTag := 'B3';
    stSDSPersistent.astGarageSlot[E_SDSGarageYStates.B4].sTag := 'B4';

    stSDSPersistent.astGarageSlot[E_SDSGarageYStates.T1].fDeg := 0.0;
    stSDSPersistent.astGarageSlot[E_SDSGarageYStates.M1].fDeg := 0.0;
    stSDSPersistent.astGarageSlot[E_SDSGarageYStates.B1].fDeg := 0.0;

    stSDSPersistent.astGarageSlot[E_SDSGarageYStates.T2].fDeg := 90.0;
    stSDSPersistent.astGarageSlot[E_SDSGarageYStates.M2].fDeg := 90.0;
    stSDSPersistent.astGarageSlot[E_SDSGarageYStates.B2].fDeg := 90.0;

    stSDSPersistent.astGarageSlot[E_SDSGarageYStates.T3].fDeg := 180.0;
    stSDSPersistent.astGarageSlot[E_SDSGarageYStates.M3].fDeg := 180.0;
    stSDSPersistent.astGarageSlot[E_SDSGarageYStates.B3].fDeg := 180.0;

    stSDSPersistent.astGarageSlot[E_SDSGarageYStates.T4].fDeg := 270.0;
    stSDSPersistent.astGarageSlot[E_SDSGarageYStates.M4].fDeg := 270.0;
    stSDSPersistent.astGarageSlot[E_SDSGarageYStates.B4].fDeg := 270.0;

    stSDSPersistent.astGarageSlot[E_SDSGarageYStates.T1].fYPos := -100.5;
    stSDSPersistent.astGarageSlot[E_SDSGarageYStates.T2].fYPos := -100.5;
    stSDSPersistent.astGarageSlot[E_SDSGarageYStates.T3].fYPos := -100.5;
    stSDSPersistent.astGarageSlot[E_SDSGarageYStates.T4].fYPos := -100.5;

    stSDSPersistent.astGarageSlot[E_SDSGarageYStates.M1].fYPos := -74.5;
    stSDSPersistent.astGarageSlot[E_SDSGarageYStates.M2].fYPos := -74.5;
    stSDSPersistent.astGarageSlot[E_SDSGarageYStates.M3].fYPos := -74.5;
    stSDSPersistent.astGarageSlot[E_SDSGarageYStates.M4].fYPos := -74.5;

    stSDSPersistent.astGarageSlot[E_SDSGarageYStates.B1].fYPos := -44.5;
    stSDSPersistent.astGarageSlot[E_SDSGarageYStates.B2].fYPos := -44.5;
    stSDSPersistent.astGarageSlot[E_SDSGarageYStates.B3].fYPos := -44.5;
    stSDSPersistent.astGarageSlot[E_SDSGarageYStates.B4].fYPos := -44.5;

    stSDSPersistent.fGarageHeightSafeFromCollision := -40.0;
    stSDSPersistent.fGarageRotationClearanceOffset := 45.0;

    stSDSPersistent.bInitialized := TRUE;
END_IF

IF NOT stSDSin.bInitialized THEN
    // Do all the required initialization for the non-persistent data of the sample delivery system.
    stSDSin.bHomingRequired := TRUE;

    fbStateSetup(stPositionState:=stDefault, bSetDefault:=TRUE);

    stSDSin.bInitialized := TRUE;
END_IF

// Update load/unloadable statuses for the garage, transfer arm, and the diffractometer.
UpdateLoadUnloadAbleStatuses(
    stSDS := stSDSin,
    stSDSP := stSDSPersistent
);

// Check if garage is above the threshold to rotate freely without fear of hitting the transfer arm.
ConfirmGarageFreeToRotate(
    stSDS := stSDSin,
    stSDSP := stSDSPersistent
);

// Control the sequencing of the sample delivery system.
StateMachine(
    stSDS := stSDSin,
    stSDSP := stSDSPersistent
);

// Update the position states
UpdatePositionStates(
    stSDS := stSDSin,
    stSDSP := stSDSPersistent
);

// Call state position function blocks.
stSDSin.fbTransferArmHPos1D(
    stMotionStage:=stSDSin.stTransferArmHStage,
    astPositionState:=stSDSin.astTransferArmHPosState,
    eEnumSet:=stSDSin.eTransferArmHStateSet,
    eEnumGet:=stSDSin.eTransferArmHStateGet,
    bEnable:=TRUE,
    stEpicsToPlc:=stSDSin.stTransferArmHEpicsToPlc,
    stPlcToEpics=>stSDSin.stTransferArmHPlcToEpics
);

stSDSin.fbTransferArmRPos1D(
    stMotionStage:=stSDSin.stTransferArmRStage,
    astPositionState:=stSDSin.astTransferArmRPosState,
    eEnumSet:=stSDSin.eTransferArmRStateSet,
    eEnumGet:=stSDSin.eTransferArmRStateGet,
    bEnable:=TRUE,
    stEpicsToPlc:=stSDSin.stTransferArmREpicsToPlc,
    stPlcToEpics=>stSDSin.stTransferArmRPlcToEpics
);

stSDSin.fbGarageYPos1D(
    stMotionStage:=stSDSin.stGarageYStage,
    astPositionState:=stSDSin.astGarageYPosState,
    eEnumSet:=stSDSin.eGarageYStateSet,
    eEnumGet:=stSDSin.eGarageYStateGet,
    bEnable:=TRUE,
    stEpicsToPlc:=stSDSin.stGarageYEpicsToPlc,
    stPlcToEpics=>stSDSin.stGarageYPlcToEpics
);

stSDSin.fbGarageRPos1D(
    stMotionStage:=stSDSin.stGarageRStage,
    astPositionState:=stSDSin.astGarageRPosState,
    eEnumSet:=stSDSin.eGarageRStateSet,
    eEnumGet:=stSDSin.eGarageRStateGet,
    bEnable:=TRUE,
    stEpicsToPlc:=stSDSin.stGarageREpicsToPlc,
    stPlcToEpics=>stSDSin.stGarageRPlcToEpics
);

// Ensure UI boolean commands are cleared after holding for one second.
stSDSin.stUISelect.bExitManualControl := FALSE;
stSDSin.stUISelect.bHomeGarage := FALSE;
stSDSin.stUISelect.bHomeTransferArm := FALSE;
stSDSin.stUISelect.bLoad := FALSE;
stSDSin.stUISelect.bLoadArmFromGarage := FALSE;
stSDSin.stUISelect.bLoadDiffractometerFromArm := FALSE;
stSDSin.stUISelect.bLoadGarageFromPort := FALSE;
stSDSin.stUISelect.bLoadUnloadGarageFromPort := FALSE;
stSDSin.stUISelect.bManualControl := FALSE;
stSDSin.stUISelect.bProceed := FALSE;
stSDSin.stUISelect.bCancel := FALSE;
stSDSin.stUISelect.bUnload := FALSE;
stSDSin.stUISelect.bUnloadArmToGarage := FALSE;
stSDSin.stUISelect.bUnloadDiffractometerToArm := FALSE;

// Align with the saved selection at the end of each cycle.
stSDSin.stUISelect.eGarageSlot := stSDSin.eSelectedGarageSlot;

ACTION ACT_CheckHomeStatus:

// ACTION - Check home status

CASE stSDSin.nHomingState OF
    0: // Initialization
        stSDSin.tonForwardHomingLimit(IN:=FALSE);
        IF stSDSin.stTransferArmHStage.nCommand = E_EpicsMotorCmd.HOME AND stSDSin.stTransferArmHStage.bBusy THEN
            stSDSin.nHomingState := stSDSin.nHomingState + 1;
        END_IF
    1: // Homing Sequence Triggered
        stSDSin.tonForwardHomingLimit(IN:=stSDSin.stTransferArmHStage.Axis.NcToPlc.SetVelo > 0,PT:=T#1s);
        IF stSDSin.stTransferArmHStage.nCommand = E_EpicsMotorCmd.HOME AND stSDSin.stTransferArmHStage.bHome THEN
            stSDSin.nHomingState := stSDSin.nHomingState + 1;
            stSDSin.tonHomingStateTimeout(IN:=FALSE);
            stSDSin.tonForwardHomingLimit(IN:=FALSE);
        ELSIF NOT stSDSin.stTransferArmHStage.bBusy THEN
            stSDSin.tonHomingStateTimeout(IN:=TRUE,PT:=T#5s);
            stSDSin.tonForwardHomingLimit(IN:=FALSE);
            IF stSDSin.tonHomingStateTimeout.Q THEN
                stSDSin.nHomingState := -1;
            END_IF
        END_IF
    2: // Homing Sequence Successful
        IF F_Limit(stSDSin.stTransferArmHStage.stAxisStatus.fActPosition, stSDSin.stTransferArmHStage.fHomePosition-0.1, stSDSin.stTransferArmHStage.fHomePosition+0.1, TRUE) THEN
            stSDSin.bHomingRequired := FALSE;
            stSDSin.nHomingState := 0;
            stSDSin.tonHomingRequiredTimeout(IN:=FALSE);
            stSDSin.tonHomingStateTimeout(IN:=FALSE);
        ELSIF NOT stSDSin.stTransferArmHStage.bBusy THEN
            stSDSin.tonHomingStateTimeout(IN:=TRUE,PT:=T#5s);
            IF stSDSin.tonHomingStateTimeout.Q THEN
                stSDSin.nHomingState := -1;
            END_IF
        END_IF
    -1: // Error Handling
        stSDSin.nHomingState := 0;
END_CASE

stSDSin.tonHomingRequiredTimeout(IN:=NOT stSDSin.bHomingRequired,PT:=stSDSin.tHomingRequiredTimeoutTime);
IF stSDSin.tonHomingRequiredTimeout.Q THEN
    stSDSin.bHomingRequired := TRUE;
END_IF
IF stSDSin.stTransferArmHStage.bHome AND F_Limit(
    fVal := stSDSin.stTransferArmHStage.Axis.NcToPlc.ActPos,
    fLLim := -0.01,
    fHLim := 0.01,
    bInclusive := TRUE) THEN
    stSDSin.bHomingRequired := FALSE;
END_IF

stSDSin.fMinUntilHomingRequired := TIME_TO_REAL(stSDSin.tonHomingRequiredTimeout.PT - stSDSin.tonHomingRequiredTimeout.ET) / 60000;

IF stSDSin.stTransferArmHStage.bExecute AND stSDSin.bHomingRequired AND stSDSin.stTransferArmHStage.fPosition > stSDSin.stTransferArmHStage.stAxisStatus.fActPosition AND
    stSDSin.stTransferArmHStage.nCommand <> E_EpicsMotorCmd.HOME THEN

    stSDSin.stTransferArmHStage.bError := TRUE;
    stSDSin.stTransferArmHStage.sCustomErrorMessage := 'Axis homing status overdue. Please home the axis.';
END_IF
END_ACTION


METHOD PRIVATE CheckCanDo2Criteria
VAR_IN_OUT
    bCanDo : BOOL;
    bCantDo : BOOL;
    sErrorMsg : T_MaxString;
END_VAR
VAR_INPUT
    b1 : BOOL;
    b2 : BOOL;
    sErrorMsgTF : T_MaxString;
    sErrorMsgFT : T_MaxString;
    sErrorMsgFF : T_MaxString;
END_VAR

bCanDo := FALSE;

IF b1 AND b2 THEN
    bCanDo := TRUE;
ELSIF b1 AND NOT b2 THEN
    bCantDo := TRUE;
    sErrorMsg := sErrorMsgTF;
ELSIF NOT b1 AND b2 THEN
    bCantDo := TRUE;
    sErrorMsg := sErrorMsgFT ;
ELSE
    bCantDo := TRUE;
    sErrorMsg := sErrorMsgFF;
END_IF
END_METHOD


METHOD PRIVATE CheckCanHomeGarage
VAR_IN_OUT
    stSDS : ST_SDS;
    stSDSP : ST_SDSPersistent;
END_VAR

stSDS.bSuccess := FALSE;

stSDS.sStatusMsg := 'Checking if garage can be homed.';

InitHomeGarage(
    stSDS := stSDS
);

IF stSDS.bGarageAboveCollisionHeight THEN
    stSDS.bSuccess := TRUE;
ELSE
    stSDS.bError := TRUE;
    stSDS.sErrorMsg := CONCAT('The garage must be above ',
        CONCAT(LREAL_TO_STRING(stSDSP.fGarageHeightSafeFromCollision),
        ' mm for the rotation axis to be homed.'));
END_IF
END_METHOD


